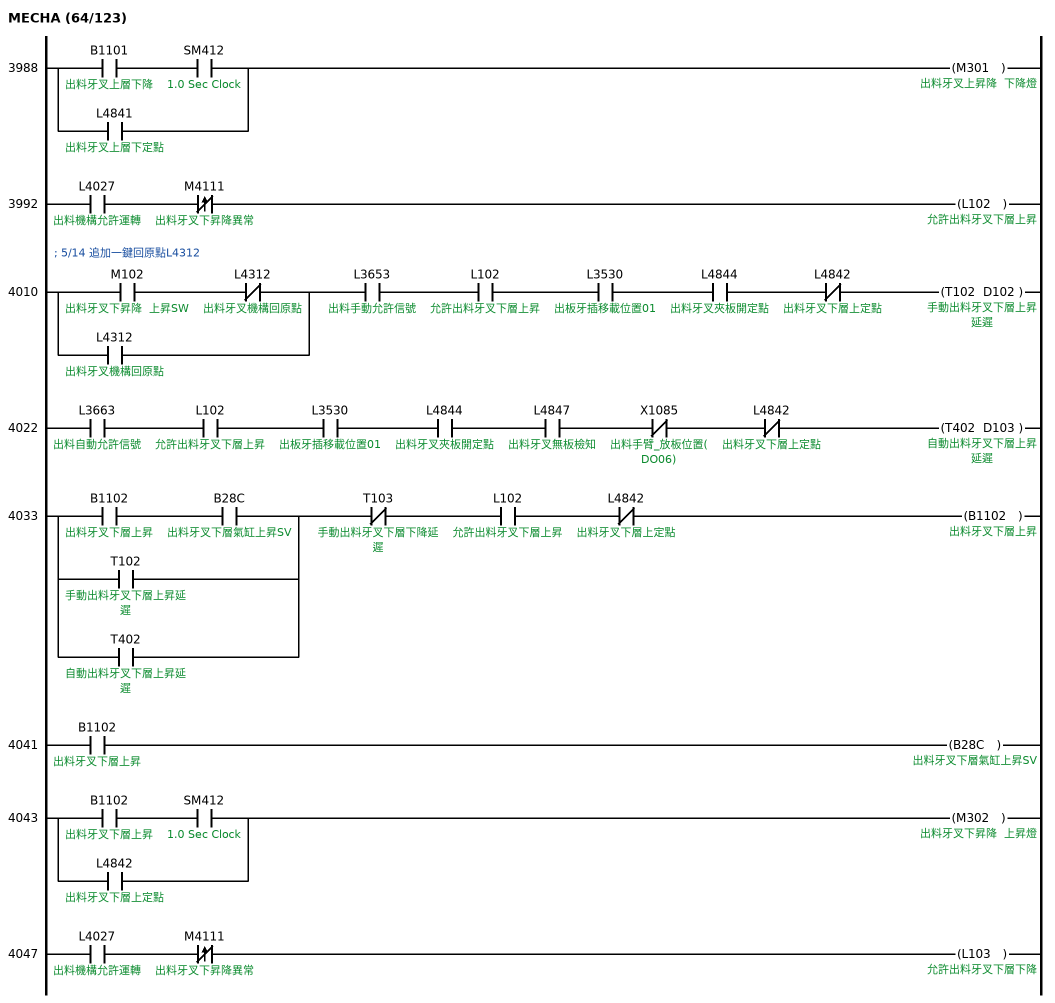
[picture p360: ladder of MECHA, rungs at steps 3988 to 4047]
3988  LD      B1101  ; 出料牙叉上層下降
      AND     SM412  ; 1.0 Sec Clock
      OR      L4841  ; 出料牙叉上層下定點
      OUT     M301  ; 出料牙叉上昇降  下降燈
3992  LD      L4027  ; 出料機構允許運轉
      ANDPI   M4111  ; 出料牙叉下昇降異常
      OUT     L102  ; 允許出料牙叉下層上昇
; 5/14 追加一鍵回原點L4312
4010  LD      M102  ; 出料牙叉下昇降  上昇SW
      ANI     L4312  ; 出料牙叉機構回原點
      OR      L4312  ; 出料牙叉機構回原點
      AND     L3653  ; 出料手動允許信號
      AND     L102  ; 允許出料牙叉下層上昇
      AND     L3530  ; 出板牙插移載位置01
      AND     L4844  ; 出料牙叉夾板開定點
      ANI     L4842  ; 出料牙叉下層上定點
      OUT     T102 D102  ; 手動出料牙叉下層上昇延遲
4022  LD      L3663  ; 出料自動允許信號
      AND     L102  ; 允許出料牙叉下層上昇
      AND     L3530  ; 出板牙插移載位置01
      AND     L4844  ; 出料牙叉夾板開定點
      AND     L4847  ; 出料牙叉無板檢知
      ANI     X1085  ; 出料手臂_放板位置(DO06)
      ANI     L4842  ; 出料牙叉下層上定點
      OUT     T402 D103  ; 自動出料牙叉下層上昇延遲
4033  LD      B1102  ; 出料牙叉下層上昇
      AND     B28C  ; 出料牙叉下層氣缸上昇SV
      OR      T102  ; 手動出料牙叉下層上昇延遲
      OR      T402  ; 自動出料牙叉下層上昇延遲
      ANI     T103  ; 手動出料牙叉下層下降延遲
      AND     L102  ; 允許出料牙叉下層上昇
      ANI     L4842  ; 出料牙叉下層上定點
      OUT     B1102  ; 出料牙叉下層上昇
4041  LD      B1102  ; 出料牙叉下層上昇
      OUT     B28C  ; 出料牙叉下層氣缸上昇SV
4043  LD      B1102  ; 出料牙叉下層上昇
      AND     SM412  ; 1.0 Sec Clock
      OR      L4842  ; 出料牙叉下層上定點
      OUT     M302  ; 出料牙叉下昇降  上昇燈
4047  LD      L4027  ; 出料機構允許運轉
      ANDPI   M4111  ; 出料牙叉下昇降異常
      OUT     L103  ; 允許出料牙叉下層下降
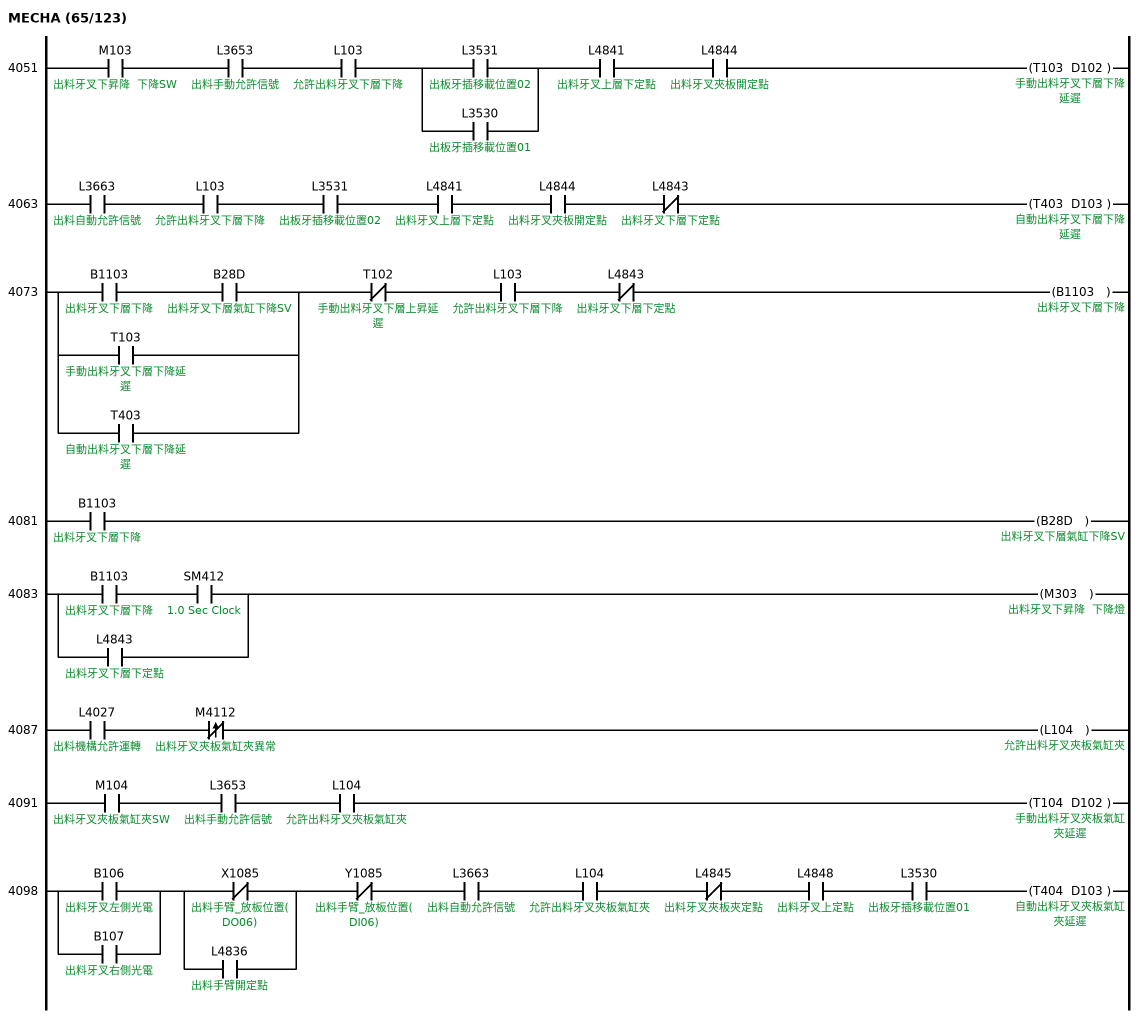
4051  LD      M103  ; 出料牙叉下昇降  下降SW
      AND     L3653  ; 出料手動允許信號
      AND     L103  ; 允許出料牙叉下層下降
      LD      L3531  ; 出板牙插移載位置02
      OR      L3530  ; 出板牙插移載位置01
      ANB
      AND     L4841  ; 出料牙叉上層下定點
      AND     L4844  ; 出料牙叉夾板開定點
      OUT     T103 D102  ; 手動出料牙叉下層下降延遲
4063  LD      L3663  ; 出料自動允許信號
      AND     L103  ; 允許出料牙叉下層下降
      AND     L3531  ; 出板牙插移載位置02
      AND     L4841  ; 出料牙叉上層下定點
      AND     L4844  ; 出料牙叉夾板開定點
      ANI     L4843  ; 出料牙叉下層下定點
      OUT     T403 D103  ; 自動出料牙叉下層下降延遲
4073  LD      B1103  ; 出料牙叉下層下降
      AND     B28D  ; 出料牙叉下層氣缸下降SV
      OR      T103  ; 手動出料牙叉下層下降延遲
      OR      T403  ; 自動出料牙叉下層下降延遲
      ANI     T102  ; 手動出料牙叉下層上昇延遲
      AND     L103  ; 允許出料牙叉下層下降
      ANI     L4843  ; 出料牙叉下層下定點
      OUT     B1103  ; 出料牙叉下層下降
4081  LD      B1103  ; 出料牙叉下層下降
      OUT     B28D  ; 出料牙叉下層氣缸下降SV
4083  LD      B1103  ; 出料牙叉下層下降
      AND     SM412  ; 1.0 Sec Clock
      OR      L4843  ; 出料牙叉下層下定點
      OUT     M303  ; 出料牙叉下昇降  下降燈
4087  LD      L4027  ; 出料機構允許運轉
      ANDPI   M4112  ; 出料牙叉夾板氣缸夾異常
      OUT     L104  ; 允許出料牙叉夾板氣缸夾
4091  LD      M104  ; 出料牙叉夾板氣缸夾SW
      AND     L3653  ; 出料手動允許信號
      AND     L104  ; 允許出料牙叉夾板氣缸夾
      OUT     T104 D102  ; 手動出料牙叉夾板氣缸夾延遲
4098  LD      B106  ; 出料牙叉左側光電
      OR      B107  ; 出料牙叉右側光電
      LDI     X1085  ; 出料手臂_放板位置(DO06)
      OR      L4836  ; 出料手臂開定點
      ANB
      ANI     Y1085  ; 出料手臂_放板位置(DI06)
      AND     L3663  ; 出料自動允許信號
      AND     L104  ; 允許出料牙叉夾板氣缸夾
      ANI     L4845  ; 出料牙叉夾板夾定點
      AND     L4848  ; 出料牙叉上定點
      AND     L3530  ; 出板牙插移載位置01
      OUT     T404 D103  ; 自動出料牙叉夾板氣缸夾延遲
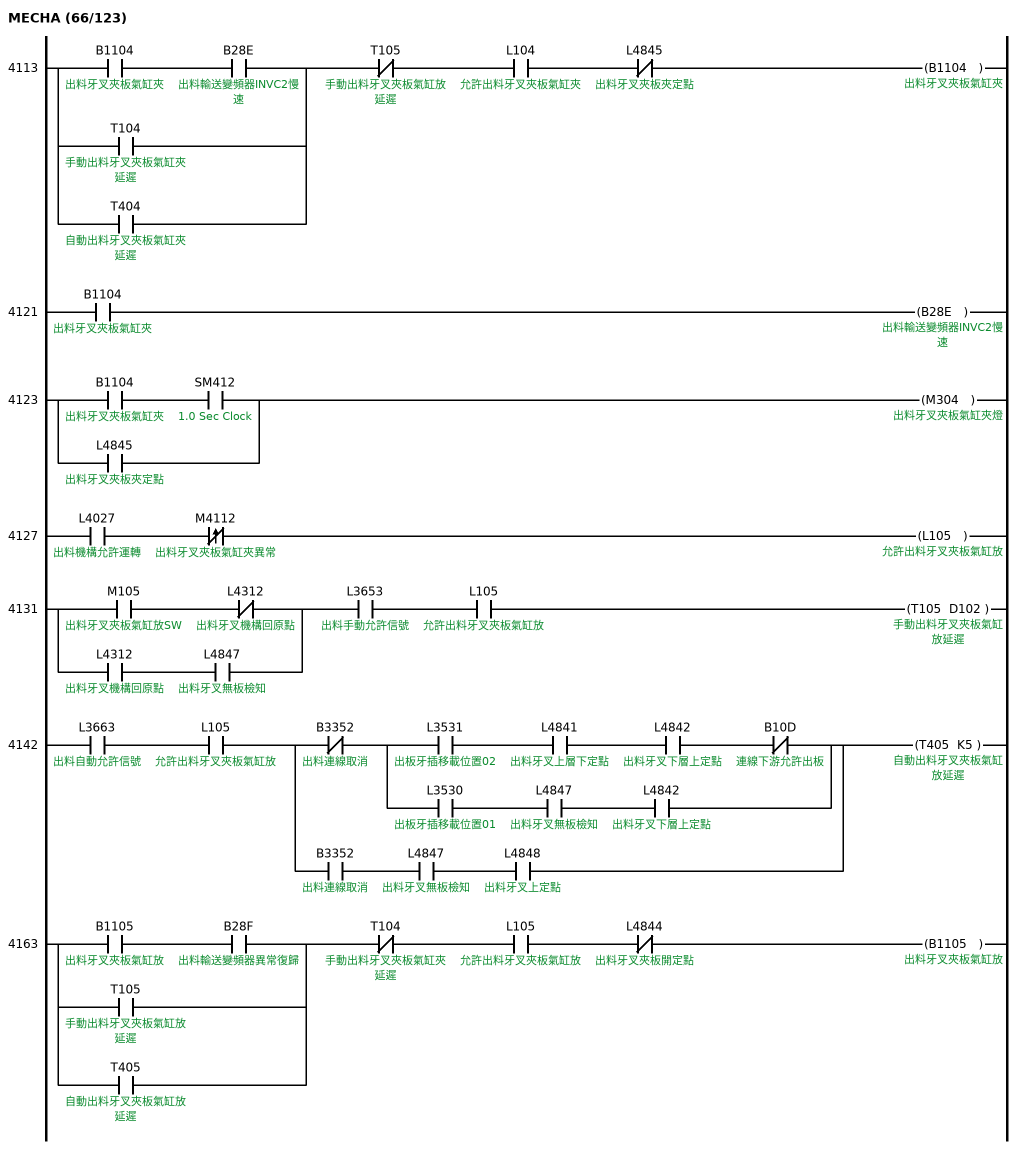
4113  LD      B1104  ; 出料牙叉夾板氣缸夾
      AND     B28E  ; 出料輸送變頻器INVC2慢速
      OR      T104  ; 手動出料牙叉夾板氣缸夾延遲
      OR      T404  ; 自動出料牙叉夾板氣缸夾延遲
      ANI     T105  ; 手動出料牙叉夾板氣缸放延遲
      AND     L104  ; 允許出料牙叉夾板氣缸夾
      ANI     L4845  ; 出料牙叉夾板夾定點
      OUT     B1104  ; 出料牙叉夾板氣缸夾
4121  LD      B1104  ; 出料牙叉夾板氣缸夾
      OUT     B28E  ; 出料輸送變頻器INVC2慢速
4123  LD      B1104  ; 出料牙叉夾板氣缸夾
      AND     SM412  ; 1.0 Sec Clock
      OR      L4845  ; 出料牙叉夾板夾定點
      OUT     M304  ; 出料牙叉夾板氣缸夾燈
4127  LD      L4027  ; 出料機構允許運轉
      ANDPI   M4112  ; 出料牙叉夾板氣缸夾異常
      OUT     L105  ; 允許出料牙叉夾板氣缸放
4131  LD      M105  ; 出料牙叉夾板氣缸放SW
      ANI     L4312  ; 出料牙叉機構回原點
      LD      L4312  ; 出料牙叉機構回原點
      AND     L4847  ; 出料牙叉無板檢知
      ORB
      AND     L3653  ; 出料手動允許信號
      AND     L105  ; 允許出料牙叉夾板氣缸放
      OUT     T105 D102  ; 手動出料牙叉夾板氣缸放延遲
4142  LD      L3663  ; 出料自動允許信號
      AND     L105  ; 允許出料牙叉夾板氣缸放
      LDI     B3352  ; 出料連線取消
      LD      L3531  ; 出板牙插移載位置02
      AND     L4841  ; 出料牙叉上層下定點
      AND     L4842  ; 出料牙叉下層上定點
      ANI     B10D  ; 連線下游允許出板
      LD      L3530  ; 出板牙插移載位置01
      AND     L4847  ; 出料牙叉無板檢知
      AND     L4842  ; 出料牙叉下層上定點
      ORB
      ANB
      LD      B3352  ; 出料連線取消
      AND     L4847  ; 出料牙叉無板檢知
      AND     L4848  ; 出料牙叉上定點
      ORB
      ANB
      OUT     T405 K5  ; 自動出料牙叉夾板氣缸放延遲
4163  LD      B1105  ; 出料牙叉夾板氣缸放
      AND     B28F  ; 出料輸送變頻器異常復歸
      OR      T105  ; 手動出料牙叉夾板氣缸放延遲
      OR      T405  ; 自動出料牙叉夾板氣缸放延遲
      ANI     T104  ; 手動出料牙叉夾板氣缸夾延遲
      AND     L105  ; 允許出料牙叉夾板氣缸放
      ANI     L4844  ; 出料牙叉夾板開定點
      OUT     B1105  ; 出料牙叉夾板氣缸放
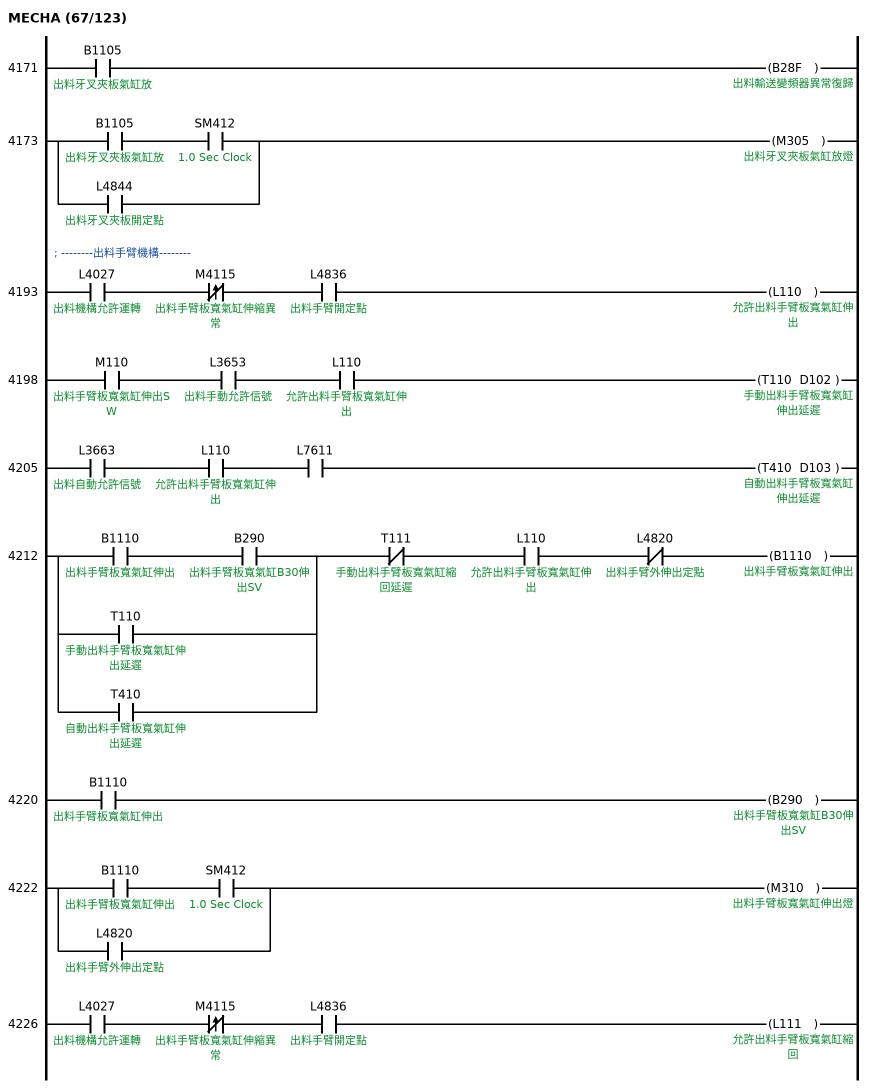
4171  LD      B1105  ; 出料牙叉夾板氣缸放
      OUT     B28F  ; 出料輸送變頻器異常復歸
4173  LD      B1105  ; 出料牙叉夾板氣缸放
      AND     SM412  ; 1.0 Sec Clock
      OR      L4844  ; 出料牙叉夾板開定點
      OUT     M305  ; 出料牙叉夾板氣缸放燈
; --------出料手臂機構--------
4193  LD      L4027  ; 出料機構允許運轉
      ANDPI   M4115  ; 出料手臂板寬氣缸伸縮異常
      AND     L4836  ; 出料手臂開定點
      OUT     L110  ; 允許出料手臂板寬氣缸伸出
4198  LD      M110  ; 出料手臂板寬氣缸伸出SW
      AND     L3653  ; 出料手動允許信號
      AND     L110  ; 允許出料手臂板寬氣缸伸出
      OUT     T110 D102  ; 手動出料手臂板寬氣缸伸出延遲
4205  LD      L3663  ; 出料自動允許信號
      AND     L110  ; 允許出料手臂板寬氣缸伸出
      AND     L7611
      OUT     T410 D103  ; 自動出料手臂板寬氣缸伸出延遲
4212  LD      B1110  ; 出料手臂板寬氣缸伸出
      AND     B290  ; 出料手臂板寬氣缸B30伸出SV
      OR      T110  ; 手動出料手臂板寬氣缸伸出延遲
      OR      T410  ; 自動出料手臂板寬氣缸伸出延遲
      ANI     T111  ; 手動出料手臂板寬氣缸縮回延遲
      AND     L110  ; 允許出料手臂板寬氣缸伸出
      ANI     L4820  ; 出料手臂外伸出定點
      OUT     B1110  ; 出料手臂板寬氣缸伸出
4220  LD      B1110  ; 出料手臂板寬氣缸伸出
      OUT     B290  ; 出料手臂板寬氣缸B30伸出SV
4222  LD      B1110  ; 出料手臂板寬氣缸伸出
      AND     SM412  ; 1.0 Sec Clock
      OR      L4820  ; 出料手臂外伸出定點
      OUT     M310  ; 出料手臂板寬氣缸伸出燈
4226  LD      L4027  ; 出料機構允許運轉
      ANDPI   M4115  ; 出料手臂板寬氣缸伸縮異常
      AND     L4836  ; 出料手臂開定點
      OUT     L111  ; 允許出料手臂板寬氣缸縮回
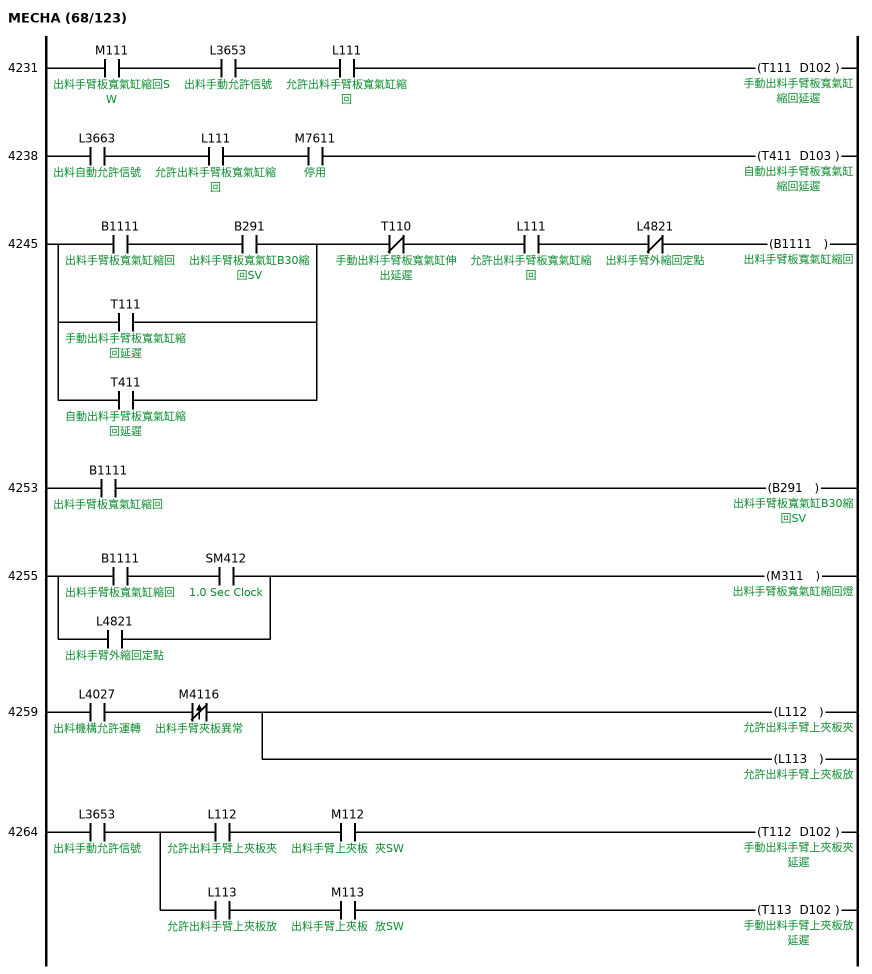
4231  LD      M111  ; 出料手臂板寬氣缸縮回SW
      AND     L3653  ; 出料手動允許信號
      AND     L111  ; 允許出料手臂板寬氣缸縮回
      OUT     T111 D102  ; 手動出料手臂板寬氣缸縮回延遲
4238  LD      L3663  ; 出料自動允許信號
      AND     L111  ; 允許出料手臂板寬氣缸縮回
      AND     M7611  ; 停用
      OUT     T411 D103  ; 自動出料手臂板寬氣缸縮回延遲
4245  LD      B1111  ; 出料手臂板寬氣缸縮回
      AND     B291  ; 出料手臂板寬氣缸B30縮回SV
      OR      T111  ; 手動出料手臂板寬氣缸縮回延遲
      OR      T411  ; 自動出料手臂板寬氣缸縮回延遲
      ANI     T110  ; 手動出料手臂板寬氣缸伸出延遲
      AND     L111  ; 允許出料手臂板寬氣缸縮回
      ANI     L4821  ; 出料手臂外縮回定點
      OUT     B1111  ; 出料手臂板寬氣缸縮回
4253  LD      B1111  ; 出料手臂板寬氣缸縮回
      OUT     B291  ; 出料手臂板寬氣缸B30縮回SV
4255  LD      B1111  ; 出料手臂板寬氣缸縮回
      AND     SM412  ; 1.0 Sec Clock
      OR      L4821  ; 出料手臂外縮回定點
      OUT     M311  ; 出料手臂板寬氣缸縮回燈
4259  LD      L4027  ; 出料機構允許運轉
      ANDPI   M4116  ; 出料手臂夾板異常
      OUT     L112  ; 允許出料手臂上夾板夾
      OUT     L113  ; 允許出料手臂上夾板放
4264  LD      L3653  ; 出料手動允許信號
      MPS
      AND     L112  ; 允許出料手臂上夾板夾
      AND     M112  ; 出料手臂上夾板  夾SW
      OUT     T112 D102  ; 手動出料手臂上夾板夾延遲
      MPP
      AND     L113  ; 允許出料手臂上夾板放
      AND     M113  ; 出料手臂上夾板  放SW
      OUT     T113 D102  ; 手動出料手臂上夾板放延遲
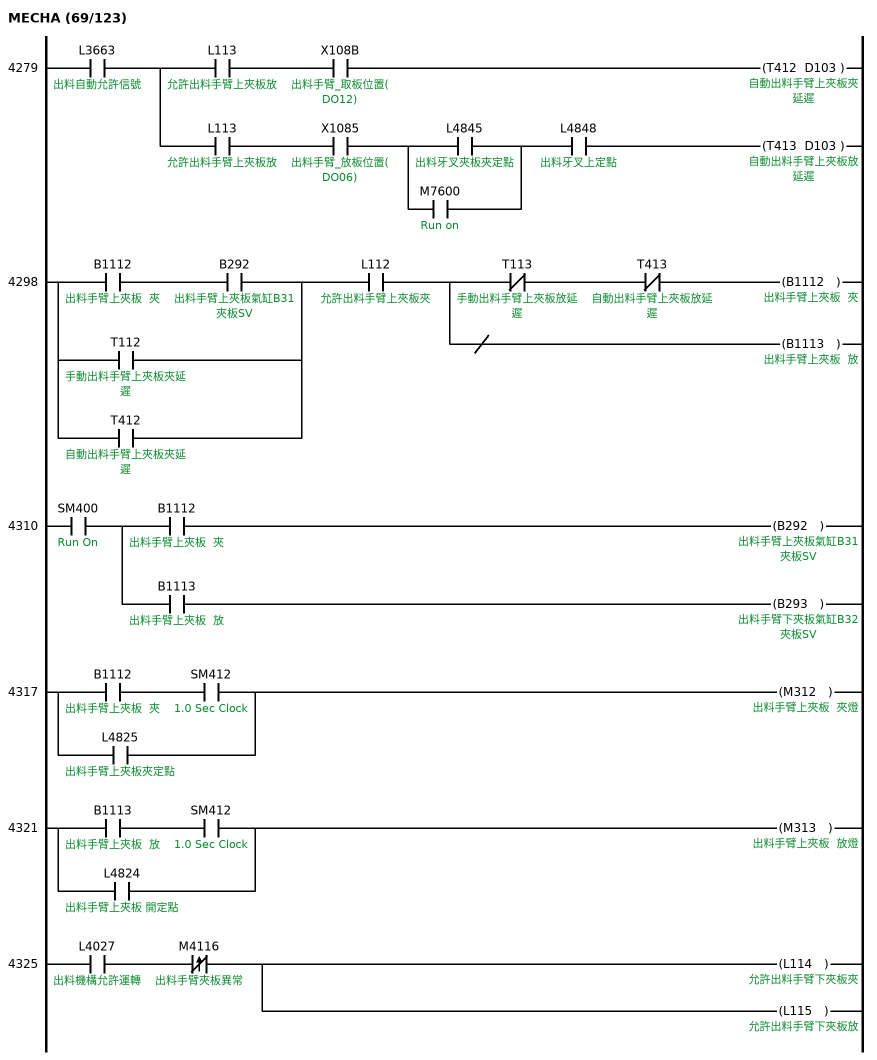
4279  LD      L3663  ; 出料自動允許信號
      MPS
      AND     L113  ; 允許出料手臂上夾板放
      AND     X108B  ; 出料手臂_取板位置(DO12)
      OUT     T412 D103  ; 自動出料手臂上夾板夾延遲
      MPP
      AND     L113  ; 允許出料手臂上夾板放
      AND     X1085  ; 出料手臂_放板位置(DO06)
      LD      L4845  ; 出料牙叉夾板夾定點
      OR      M7600  ; Run on
      ANB
      AND     L4848  ; 出料牙叉上定點
      OUT     T413 D103  ; 自動出料手臂上夾板放延遲
4298  LD      B1112  ; 出料手臂上夾板  夾
      AND     B292  ; 出料手臂上夾板氣缸B31夾板SV
      OR      T112  ; 手動出料手臂上夾板夾延遲
      OR      T412  ; 自動出料手臂上夾板夾延遲
      AND     L112  ; 允許出料手臂上夾板夾
      MPS
      ANI     T113  ; 手動出料手臂上夾板放延遲
      ANI     T413  ; 自動出料手臂上夾板放延遲
      OUT     B1112  ; 出料手臂上夾板  夾
      MPP
      INV
      OUT     B1113  ; 出料手臂上夾板  放
4310  LD      SM400  ; Run On
      MPS
      AND     B1112  ; 出料手臂上夾板  夾
      OUT     B292  ; 出料手臂上夾板氣缸B31夾板SV
      MPP
      AND     B1113  ; 出料手臂上夾板  放
      OUT     B293  ; 出料手臂下夾板氣缸B32夾板SV
4317  LD      B1112  ; 出料手臂上夾板  夾
      AND     SM412  ; 1.0 Sec Clock
      OR      L4825  ; 出料手臂上夾板夾定點
      OUT     M312  ; 出料手臂上夾板  夾燈
4321  LD      B1113  ; 出料手臂上夾板  放
      AND     SM412  ; 1.0 Sec Clock
      OR      L4824  ; 出料手臂上夾板 開定點
      OUT     M313  ; 出料手臂上夾板  放燈
4325  LD      L4027  ; 出料機構允許運轉
      ANDPI   M4116  ; 出料手臂夾板異常
      OUT     L114  ; 允許出料手臂下夾板夾
      OUT     L115  ; 允許出料手臂下夾板放
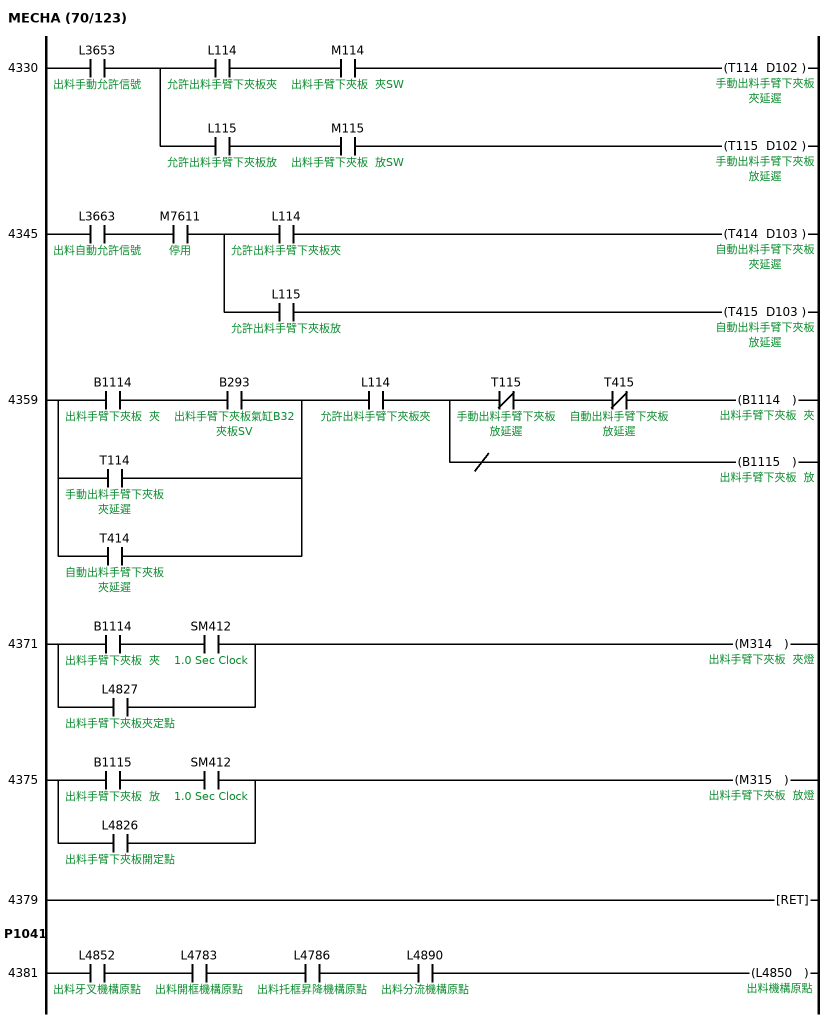
4330  LD      L3653  ; 出料手動允許信號
      MPS
      AND     L114  ; 允許出料手臂下夾板夾
      AND     M114  ; 出料手臂下夾板  夾SW
      OUT     T114 D102  ; 手動出料手臂下夾板  夾延遲
      MPP
      AND     L115  ; 允許出料手臂下夾板放
      AND     M115  ; 出料手臂下夾板  放SW
      OUT     T115 D102  ; 手動出料手臂下夾板  放延遲
4345  LD      L3663  ; 出料自動允許信號
      AND     M7611  ; 停用
      MPS
      AND     L114  ; 允許出料手臂下夾板夾
      OUT     T414 D103  ; 自動出料手臂下夾板  夾延遲
      MPP
      AND     L115  ; 允許出料手臂下夾板放
      OUT     T415 D103  ; 自動出料手臂下夾板  放延遲
4359  LD      B1114  ; 出料手臂下夾板  夾
      AND     B293  ; 出料手臂下夾板氣缸B32夾板SV
      OR      T114  ; 手動出料手臂下夾板  夾延遲
      OR      T414  ; 自動出料手臂下夾板  夾延遲
      AND     L114  ; 允許出料手臂下夾板夾
      MPS
      ANI     T115  ; 手動出料手臂下夾板  放延遲
      ANI     T415  ; 自動出料手臂下夾板  放延遲
      OUT     B1114  ; 出料手臂下夾板  夾
      MPP
      INV
      OUT     B1115  ; 出料手臂下夾板  放
4371  LD      B1114  ; 出料手臂下夾板  夾
      AND     SM412  ; 1.0 Sec Clock
      OR      L4827  ; 出料手臂下夾板夾定點
      OUT     M314  ; 出料手臂下夾板  夾燈
4375  LD      B1115  ; 出料手臂下夾板  放
      AND     SM412  ; 1.0 Sec Clock
      OR      L4826  ; 出料手臂下夾板開定點
      OUT     M315  ; 出料手臂下夾板  放燈
4379  RET
      P1041
4381  LD      L4852  ; 出料牙叉機構原點
      AND     L4783  ; 出料開框機構原點
      AND     L4786  ; 出料托框昇降機構原點
      AND     L4890  ; 出料分流機構原點
      OUT     L4850  ; 出料機構原點
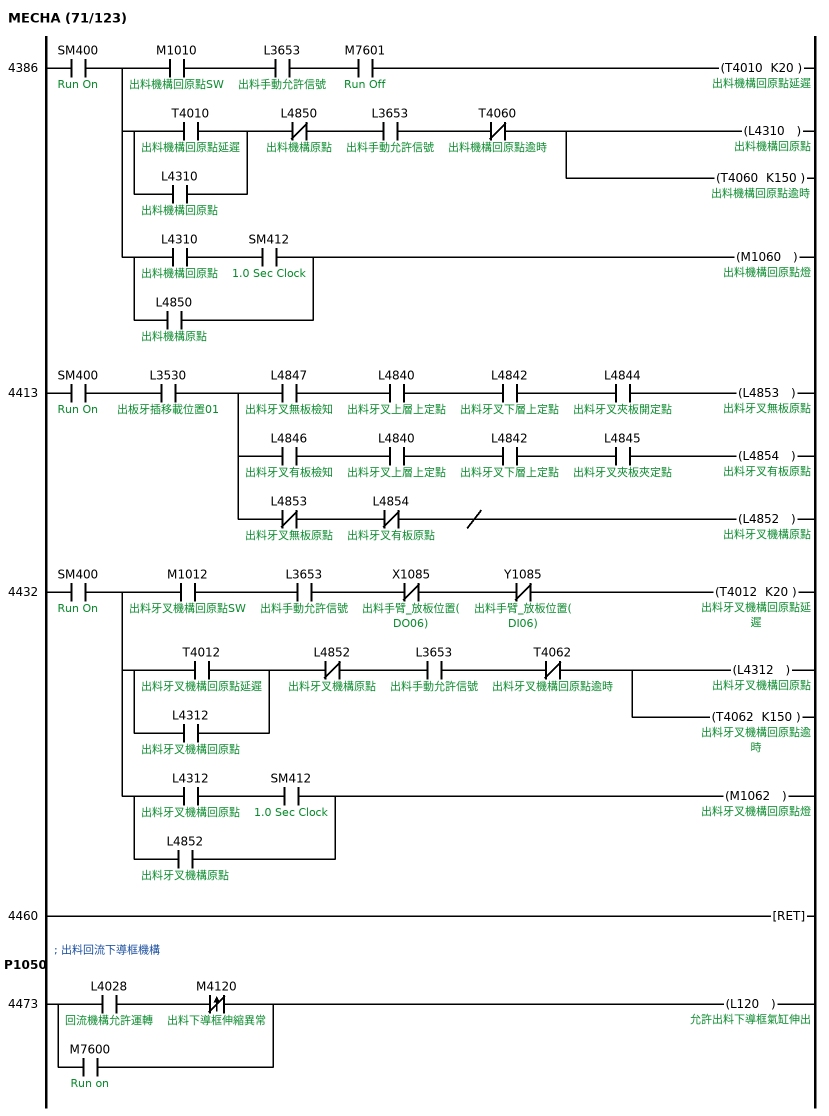
4386  LD      SM400  ; Run On
      MPS
      AND     M1010  ; 出料機構回原點SW
      AND     L3653  ; 出料手動允許信號
      AND     M7601  ; Run Off
      OUT     T4010 K20  ; 出料機構回原點延遲
      MRD
      LD      T4010  ; 出料機構回原點延遲
      OR      L4310  ; 出料機構回原點
      ANB
      ANI     L4850  ; 出料機構原點
      AND     L3653  ; 出料手動允許信號
      ANI     T4060  ; 出料機構回原點逾時
      OUT     L4310  ; 出料機構回原點
      OUT     T4060 K150  ; 出料機構回原點逾時
      MPP
      LD      L4310  ; 出料機構回原點
      AND     SM412  ; 1.0 Sec Clock
      OR      L4850  ; 出料機構原點
      ANB
      OUT     M1060  ; 出料機構回原點燈
4413  LD      SM400  ; Run On
      AND     L3530  ; 出板牙插移載位置01
      MPS
      AND     L4847  ; 出料牙叉無板檢知
      AND     L4840  ; 出料牙叉上層上定點
      AND     L4842  ; 出料牙叉下層上定點
      AND     L4844  ; 出料牙叉夾板開定點
      OUT     L4853  ; 出料牙叉無板原點
      MRD
      AND     L4846  ; 出料牙叉有板檢知
      AND     L4840  ; 出料牙叉上層上定點
      AND     L4842  ; 出料牙叉下層上定點
      AND     L4845  ; 出料牙叉夾板夾定點
      OUT     L4854  ; 出料牙叉有板原點
      MPP
      ANI     L4853  ; 出料牙叉無板原點
      ANI     L4854  ; 出料牙叉有板原點
      INV
      OUT     L4852  ; 出料牙叉機構原點
4432  LD      SM400  ; Run On
      MPS
      AND     M1012  ; 出料牙叉機構回原點SW
      AND     L3653  ; 出料手動允許信號
      ANI     X1085  ; 出料手臂_放板位置(DO06)
      ANI     Y1085  ; 出料手臂_放板位置(DI06)
      OUT     T4012 K20  ; 出料牙叉機構回原點延遲
      MRD
      LD      T4012  ; 出料牙叉機構回原點延遲
      OR      L4312  ; 出料牙叉機構回原點
      ANB
      ANI     L4852  ; 出料牙叉機構原點
      AND     L3653  ; 出料手動允許信號
      ANI     T4062  ; 出料牙叉機構回原點逾時
      OUT     L4312  ; 出料牙叉機構回原點
      OUT     T4062 K150  ; 出料牙叉機構回原點逾時
      MPP
      LD      L4312  ; 出料牙叉機構回原點
      AND     SM412  ; 1.0 Sec Clock
      OR      L4852  ; 出料牙叉機構原點
      ANB
      OUT     M1062  ; 出料牙叉機構回原點燈
4460  RET
; 出料回流下導框機構
      P1050
4473  LD      L4028  ; 回流機構允許運轉
      ANDPI   M4120  ; 出料下導框伸縮異常
      OR      M7600  ; Run on
      OUT     L120  ; 允許出料下導框氣缸伸出
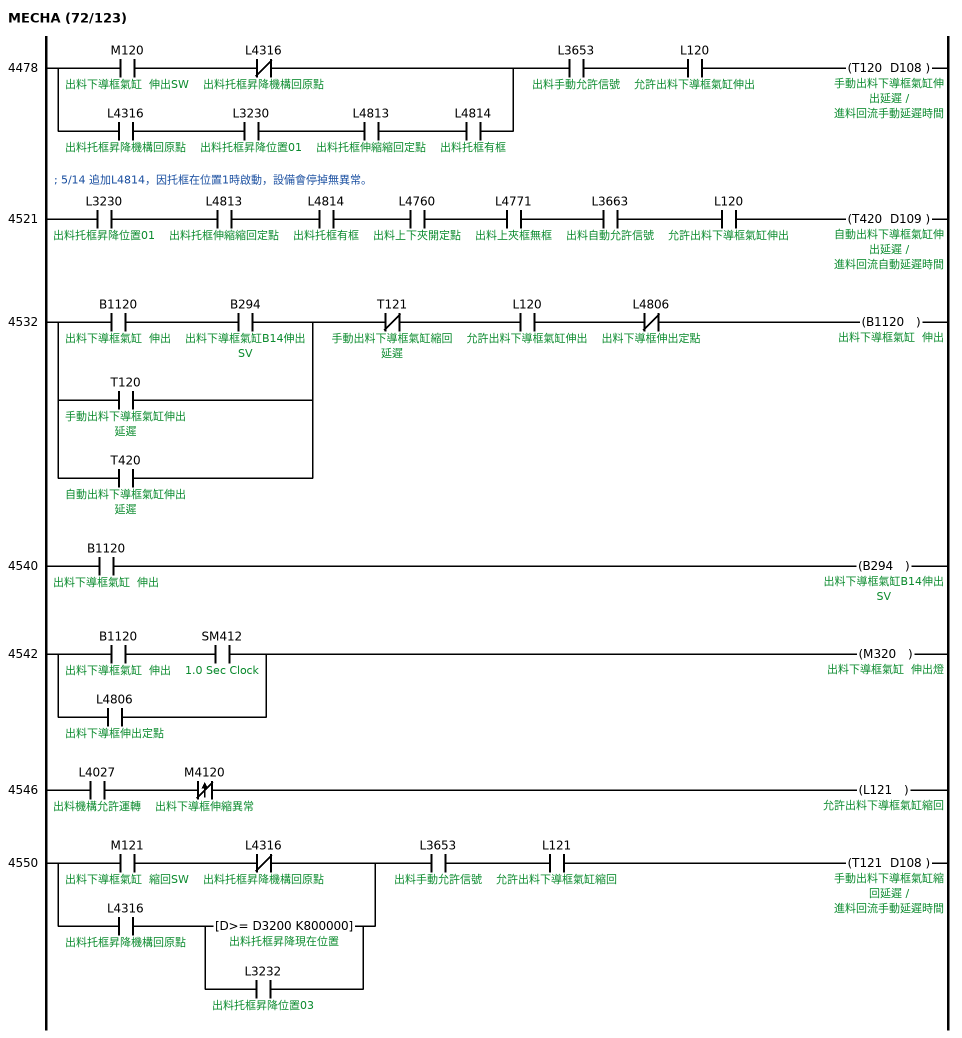
4478  LD      M120  ; 出料下導框氣缸  伸出SW
      ANI     L4316  ; 出料托框昇降機構回原點
      LD      L4316  ; 出料托框昇降機構回原點
      AND     L3230  ; 出料托框昇降位置01
      AND     L4813  ; 出料托框伸縮縮回定點
      AND     L4814  ; 出料托框有框
      ORB
      AND     L3653  ; 出料手動允許信號
      AND     L120  ; 允許出料下導框氣缸伸出
      OUT     T120 D108  ; 手動出料下導框氣缸伸出延遲 / 進料回流手動延遲時間
; 5/14 追加L4814，因托框在位置1時啟動，設備會停掉無異常。
4521  LD      L3230  ; 出料托框昇降位置01
      AND     L4813  ; 出料托框伸縮縮回定點
      AND     L4814  ; 出料托框有框
      AND     L4760  ; 出料上下夾開定點
      AND     L4771  ; 出料上夾框無框
      AND     L3663  ; 出料自動允許信號
      AND     L120  ; 允許出料下導框氣缸伸出
      OUT     T420 D109  ; 自動出料下導框氣缸伸出延遲 / 進料回流自動延遲時間
4532  LD      B1120  ; 出料下導框氣缸  伸出
      AND     B294  ; 出料下導框氣缸B14伸出SV
      OR      T120  ; 手動出料下導框氣缸伸出延遲
      OR      T420  ; 自動出料下導框氣缸伸出延遲
      ANI     T121  ; 手動出料下導框氣缸縮回延遲
      AND     L120  ; 允許出料下導框氣缸伸出
      ANI     L4806  ; 出料下導框伸出定點
      OUT     B1120  ; 出料下導框氣缸  伸出
4540  LD      B1120  ; 出料下導框氣缸  伸出
      OUT     B294  ; 出料下導框氣缸B14伸出SV
4542  LD      B1120  ; 出料下導框氣缸  伸出
      AND     SM412  ; 1.0 Sec Clock
      OR      L4806  ; 出料下導框伸出定點
      OUT     M320  ; 出料下導框氣缸  伸出燈
4546  LD      L4027  ; 出料機構允許運轉
      ANDPI   M4120  ; 出料下導框伸縮異常
      OUT     L121  ; 允許出料下導框氣缸縮回
4550  LD      M121  ; 出料下導框氣缸  縮回SW
      ANI     L4316  ; 出料托框昇降機構回原點
      LD      L4316  ; 出料托框昇降機構回原點
      LDD>=   D3200 K800000  ; 出料托框昇降現在位置
      OR      L3232  ; 出料托框昇降位置03
      ANB
      ORB
      AND     L3653  ; 出料手動允許信號
      AND     L121  ; 允許出料下導框氣缸縮回
      OUT     T121 D108  ; 手動出料下導框氣缸縮回延遲 / 進料回流手動延遲時間
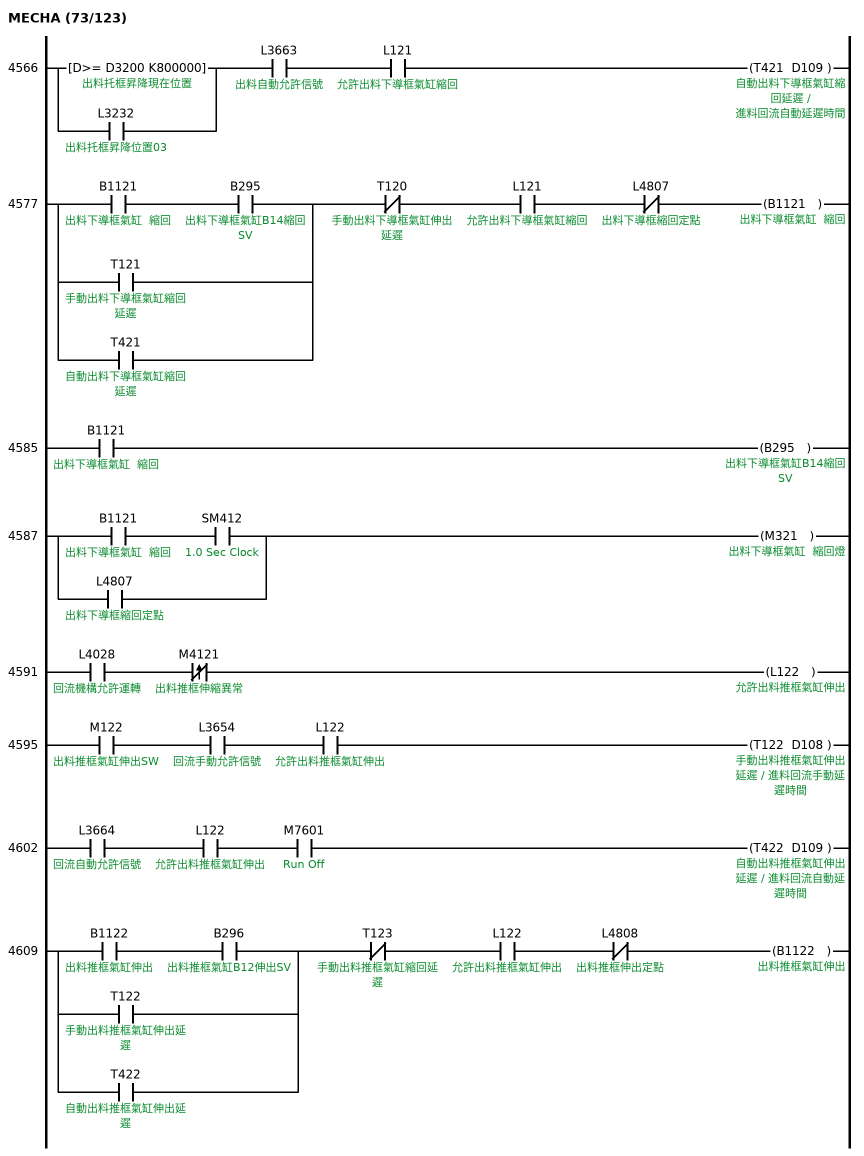
4566  LDD>=   D3200 K800000  ; 出料托框昇降現在位置
      OR      L3232  ; 出料托框昇降位置03
      AND     L3663  ; 出料自動允許信號
      AND     L121  ; 允許出料下導框氣缸縮回
      OUT     T421 D109  ; 自動出料下導框氣缸縮回延遲 / 進料回流自動延遲時間
4577  LD      B1121  ; 出料下導框氣缸  縮回
      AND     B295  ; 出料下導框氣缸B14縮回SV
      OR      T121  ; 手動出料下導框氣缸縮回延遲
      OR      T421  ; 自動出料下導框氣缸縮回延遲
      ANI     T120  ; 手動出料下導框氣缸伸出延遲
      AND     L121  ; 允許出料下導框氣缸縮回
      ANI     L4807  ; 出料下導框縮回定點
      OUT     B1121  ; 出料下導框氣缸  縮回
4585  LD      B1121  ; 出料下導框氣缸  縮回
      OUT     B295  ; 出料下導框氣缸B14縮回SV
4587  LD      B1121  ; 出料下導框氣缸  縮回
      AND     SM412  ; 1.0 Sec Clock
      OR      L4807  ; 出料下導框縮回定點
      OUT     M321  ; 出料下導框氣缸  縮回燈
4591  LD      L4028  ; 回流機構允許運轉
      ANDPI   M4121  ; 出料推框伸縮異常
      OUT     L122  ; 允許出料推框氣缸伸出
4595  LD      M122  ; 出料推框氣缸伸出SW
      AND     L3654  ; 回流手動允許信號
      AND     L122  ; 允許出料推框氣缸伸出
      OUT     T122 D108  ; 手動出料推框氣缸伸出延遲 / 進料回流手動延遲時間
4602  LD      L3664  ; 回流自動允許信號
      AND     L122  ; 允許出料推框氣缸伸出
      AND     M7601  ; Run Off
      OUT     T422 D109  ; 自動出料推框氣缸伸出延遲 / 進料回流自動延遲時間
4609  LD      B1122  ; 出料推框氣缸伸出
      AND     B296  ; 出料推框氣缸B12伸出SV
      OR      T122  ; 手動出料推框氣缸伸出延遲
      OR      T422  ; 自動出料推框氣缸伸出延遲
      ANI     T123  ; 手動出料推框氣缸縮回延遲
      AND     L122  ; 允許出料推框氣缸伸出
      ANI     L4808  ; 出料推框伸出定點
      OUT     B1122  ; 出料推框氣缸伸出
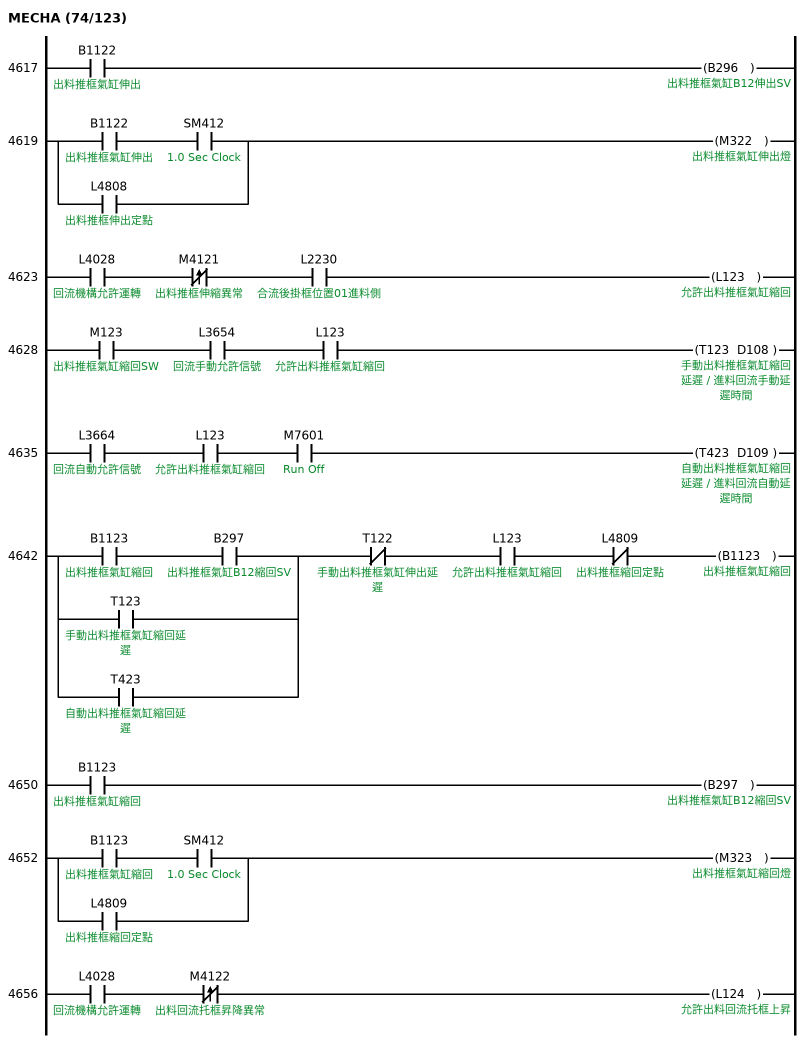
4617  LD      B1122  ; 出料推框氣缸伸出
      OUT     B296  ; 出料推框氣缸B12伸出SV
4619  LD      B1122  ; 出料推框氣缸伸出
      AND     SM412  ; 1.0 Sec Clock
      OR      L4808  ; 出料推框伸出定點
      OUT     M322  ; 出料推框氣缸伸出燈
4623  LD      L4028  ; 回流機構允許運轉
      ANDPI   M4121  ; 出料推框伸縮異常
      AND     L2230  ; 合流後掛框位置01進料側
      OUT     L123  ; 允許出料推框氣缸縮回
4628  LD      M123  ; 出料推框氣缸縮回SW
      AND     L3654  ; 回流手動允許信號
      AND     L123  ; 允許出料推框氣缸縮回
      OUT     T123 D108  ; 手動出料推框氣缸縮回延遲 / 進料回流手動延遲時間
4635  LD      L3664  ; 回流自動允許信號
      AND     L123  ; 允許出料推框氣缸縮回
      AND     M7601  ; Run Off
      OUT     T423 D109  ; 自動出料推框氣缸縮回延遲 / 進料回流自動延遲時間
4642  LD      B1123  ; 出料推框氣缸縮回
      AND     B297  ; 出料推框氣缸B12縮回SV
      OR      T123  ; 手動出料推框氣缸縮回延遲
      OR      T423  ; 自動出料推框氣缸縮回延遲
      ANI     T122  ; 手動出料推框氣缸伸出延遲
      AND     L123  ; 允許出料推框氣缸縮回
      ANI     L4809  ; 出料推框縮回定點
      OUT     B1123  ; 出料推框氣缸縮回
4650  LD      B1123  ; 出料推框氣缸縮回
      OUT     B297  ; 出料推框氣缸B12縮回SV
4652  LD      B1123  ; 出料推框氣缸縮回
      AND     SM412  ; 1.0 Sec Clock
      OR      L4809  ; 出料推框縮回定點
      OUT     M323  ; 出料推框氣缸縮回燈
4656  LD      L4028  ; 回流機構允許運轉
      ANDPI   M4122  ; 出料回流托框昇降異常
      OUT     L124  ; 允許出料回流托框上昇
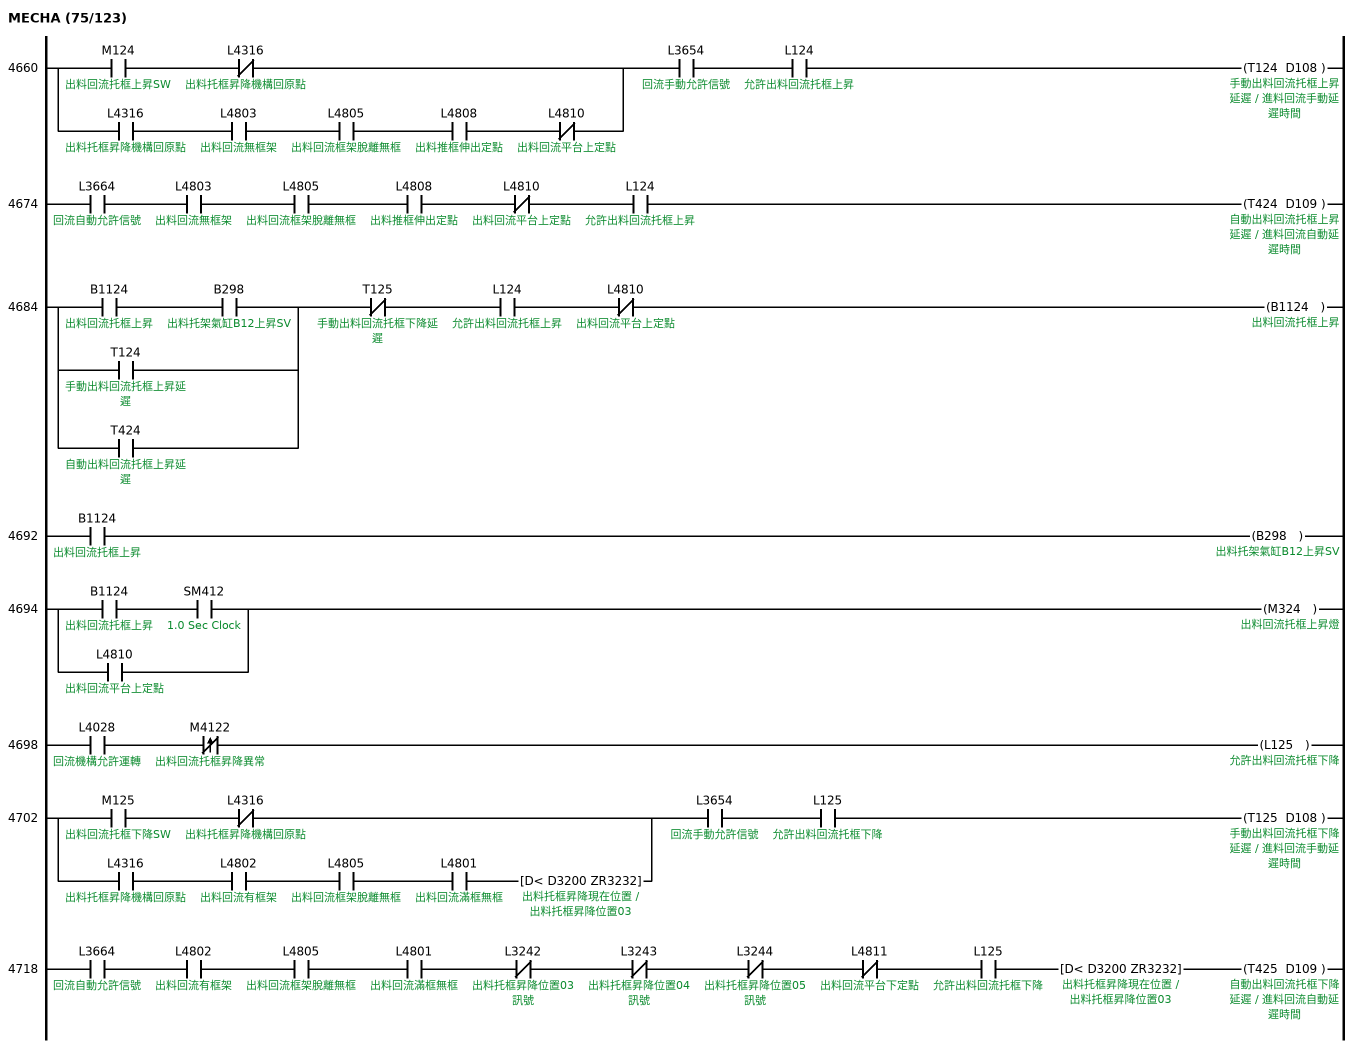
4660  LD      M124  ; 出料回流托框上昇SW
      ANI     L4316  ; 出料托框昇降機構回原點
      LD      L4316  ; 出料托框昇降機構回原點
      AND     L4803  ; 出料回流無框架
      AND     L4805  ; 出料回流框架脫離無框
      AND     L4808  ; 出料推框伸出定點
      ANI     L4810  ; 出料回流平台上定點
      ORB
      AND     L3654  ; 回流手動允許信號
      AND     L124  ; 允許出料回流托框上昇
      OUT     T124 D108  ; 手動出料回流托框上昇延遲 / 進料回流手動延遲時間
4674  LD      L3664  ; 回流自動允許信號
      AND     L4803  ; 出料回流無框架
      AND     L4805  ; 出料回流框架脫離無框
      AND     L4808  ; 出料推框伸出定點
      ANI     L4810  ; 出料回流平台上定點
      AND     L124  ; 允許出料回流托框上昇
      OUT     T424 D109  ; 自動出料回流托框上昇延遲 / 進料回流自動延遲時間
4684  LD      B1124  ; 出料回流托框上昇
      AND     B298  ; 出料托架氣缸B12上昇SV
      OR      T124  ; 手動出料回流托框上昇延遲
      OR      T424  ; 自動出料回流托框上昇延遲
      ANI     T125  ; 手動出料回流托框下降延遲
      AND     L124  ; 允許出料回流托框上昇
      ANI     L4810  ; 出料回流平台上定點
      OUT     B1124  ; 出料回流托框上昇
4692  LD      B1124  ; 出料回流托框上昇
      OUT     B298  ; 出料托架氣缸B12上昇SV
4694  LD      B1124  ; 出料回流托框上昇
      AND     SM412  ; 1.0 Sec Clock
      OR      L4810  ; 出料回流平台上定點
      OUT     M324  ; 出料回流托框上昇燈
4698  LD      L4028  ; 回流機構允許運轉
      ANDPI   M4122  ; 出料回流托框昇降異常
      OUT     L125  ; 允許出料回流托框下降
4702  LD      M125  ; 出料回流托框下降SW
      ANI     L4316  ; 出料托框昇降機構回原點
      LD      L4316  ; 出料托框昇降機構回原點
      AND     L4802  ; 出料回流有框架
      AND     L4805  ; 出料回流框架脫離無框
      AND     L4801  ; 出料回流滿框無框
      ANDD<   D3200 ZR3232  ; 出料托框昇降現在位置 / 出料托框昇降位置03
      ORB
      AND     L3654  ; 回流手動允許信號
      AND     L125  ; 允許出料回流托框下降
      OUT     T125 D108  ; 手動出料回流托框下降延遲 / 進料回流手動延遲時間
4718  LD      L3664  ; 回流自動允許信號
      AND     L4802  ; 出料回流有框架
      AND     L4805  ; 出料回流框架脫離無框
      AND     L4801  ; 出料回流滿框無框
      ANI     L3242  ; 出料托框昇降位置03 訊號
      ANI     L3243  ; 出料托框昇降位置04 訊號
      ANI     L3244  ; 出料托框昇降位置05 訊號
      ANI     L4811  ; 出料回流平台下定點
      AND     L125  ; 允許出料回流托框下降
      ANDD<   D3200 ZR3232  ; 出料托框昇降現在位置 / 出料托框昇降位置03
      OUT     T425 D109  ; 自動出料回流托框下降延遲 / 進料回流自動延遲時間
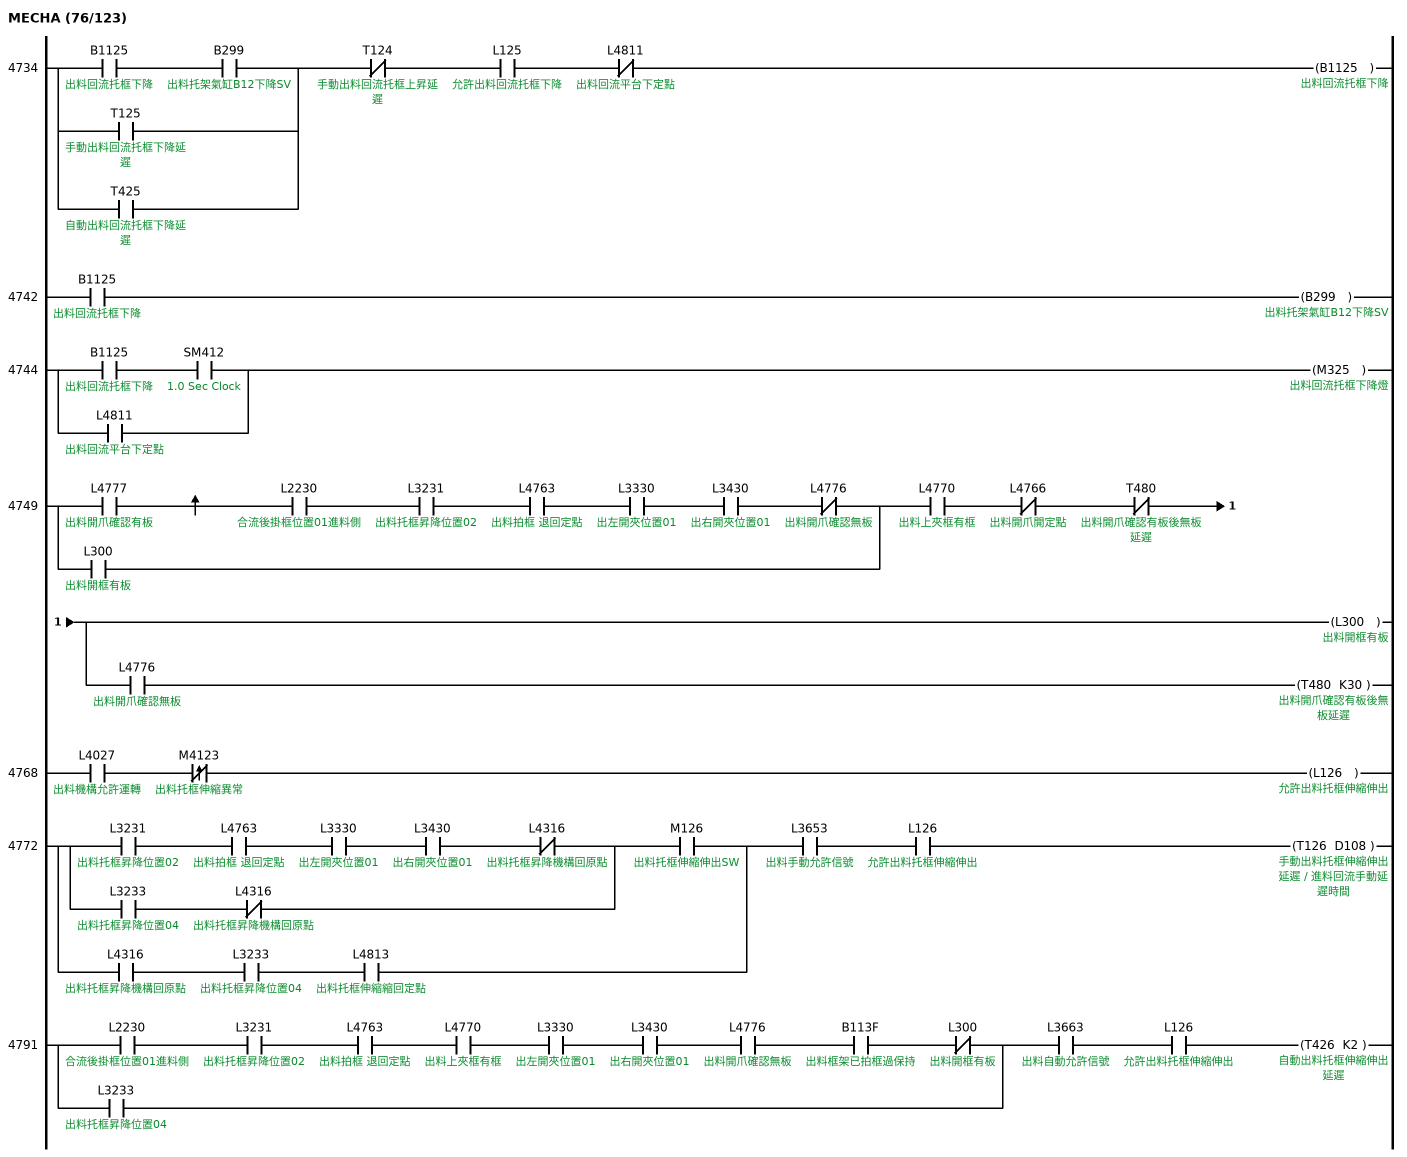
4734  LD      B1125  ; 出料回流托框下降
      AND     B299  ; 出料托架氣缸B12下降SV
      OR      T125  ; 手動出料回流托框下降延遲
      OR      T425  ; 自動出料回流托框下降延遲
      ANI     T124  ; 手動出料回流托框上昇延遲
      AND     L125  ; 允許出料回流托框下降
      ANI     L4811  ; 出料回流平台下定點
      OUT     B1125  ; 出料回流托框下降
4742  LD      B1125  ; 出料回流托框下降
      OUT     B299  ; 出料托架氣缸B12下降SV
4744  LD      B1125  ; 出料回流托框下降
      AND     SM412  ; 1.0 Sec Clock
      OR      L4811  ; 出料回流平台下定點
      OUT     M325  ; 出料回流托框下降燈
4749  LD      L4777  ; 出料開爪確認有板
      MEP
      AND     L2230  ; 合流後掛框位置01進料側
      AND     L3231  ; 出料托框昇降位置02
      AND     L4763  ; 出料拍框 退回定點
      AND     L3330  ; 出左開夾位置01
      AND     L3430  ; 出右開夾位置01
      ANI     L4776  ; 出料開爪確認無板
      OR      L300  ; 出料開框有板
      AND     L4770  ; 出料上夾框有框
      ANI     L4766  ; 出料開爪開定點
      ANI     T480  ; 出料開爪確認有板後無板延遲
      OUT     L300  ; 出料開框有板
      AND     L4776  ; 出料開爪確認無板
      OUT     T480 K30  ; 出料開爪確認有板後無板延遲
4768  LD      L4027  ; 出料機構允許運轉
      ANDPI   M4123  ; 出料托框伸縮異常
      OUT     L126  ; 允許出料托框伸縮伸出
4772  LD      L3231  ; 出料托框昇降位置02
      AND     L4763  ; 出料拍框 退回定點
      AND     L3330  ; 出左開夾位置01
      AND     L3430  ; 出右開夾位置01
      ANI     L4316  ; 出料托框昇降機構回原點
      LD      L3233  ; 出料托框昇降位置04
      ANI     L4316  ; 出料托框昇降機構回原點
      ORB
      AND     M126  ; 出料托框伸縮伸出SW
      LD      L4316  ; 出料托框昇降機構回原點
      AND     L3233  ; 出料托框昇降位置04
      AND     L4813  ; 出料托框伸縮縮回定點
      ORB
      AND     L3653  ; 出料手動允許信號
      AND     L126  ; 允許出料托框伸縮伸出
      OUT     T126 D108  ; 手動出料托框伸縮伸出延遲 / 進料回流手動延遲時間
4791  LD      L2230  ; 合流後掛框位置01進料側
      AND     L3231  ; 出料托框昇降位置02
      AND     L4763  ; 出料拍框 退回定點
      AND     L4770  ; 出料上夾框有框
      AND     L3330  ; 出左開夾位置01
      AND     L3430  ; 出右開夾位置01
      AND     L4776  ; 出料開爪確認無板
      AND     B113F  ; 出料框架已拍框過保持
      ANI     L300  ; 出料開框有板
      OR      L3233  ; 出料托框昇降位置04
      AND     L3663  ; 出料自動允許信號
      AND     L126  ; 允許出料托框伸縮伸出
      OUT     T426 K2  ; 自動出料托框伸縮伸出延遲
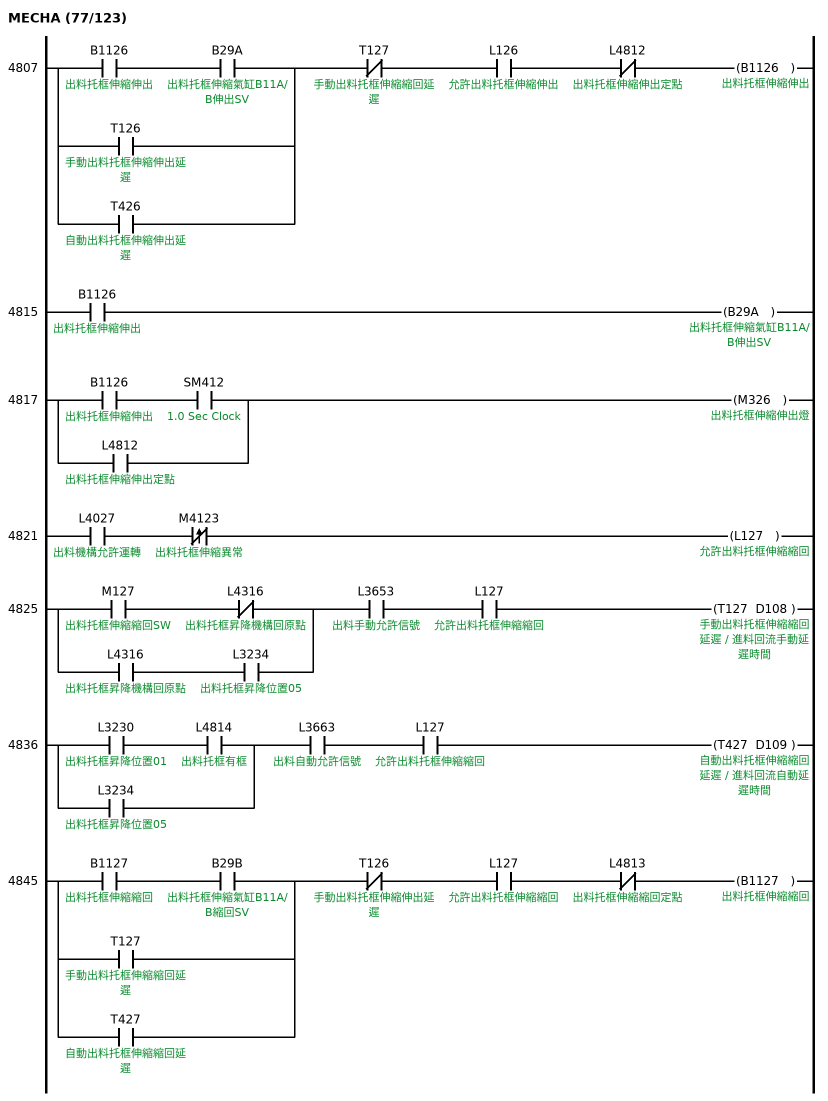
4807  LD      B1126  ; 出料托框伸縮伸出
      AND     B29A  ; 出料托框伸縮氣缸B11A/B伸出SV
      OR      T126  ; 手動出料托框伸縮伸出延遲
      OR      T426  ; 自動出料托框伸縮伸出延遲
      ANI     T127  ; 手動出料托框伸縮縮回延遲
      AND     L126  ; 允許出料托框伸縮伸出
      ANI     L4812  ; 出料托框伸縮伸出定點
      OUT     B1126  ; 出料托框伸縮伸出
4815  LD      B1126  ; 出料托框伸縮伸出
      OUT     B29A  ; 出料托框伸縮氣缸B11A/B伸出SV
4817  LD      B1126  ; 出料托框伸縮伸出
      AND     SM412  ; 1.0 Sec Clock
      OR      L4812  ; 出料托框伸縮伸出定點
      OUT     M326  ; 出料托框伸縮伸出燈
4821  LD      L4027  ; 出料機構允許運轉
      ANDPI   M4123  ; 出料托框伸縮異常
      OUT     L127  ; 允許出料托框伸縮縮回
4825  LD      M127  ; 出料托框伸縮縮回SW
      ANI     L4316  ; 出料托框昇降機構回原點
      LD      L4316  ; 出料托框昇降機構回原點
      AND     L3234  ; 出料托框昇降位置05
      ORB
      AND     L3653  ; 出料手動允許信號
      AND     L127  ; 允許出料托框伸縮縮回
      OUT     T127 D108  ; 手動出料托框伸縮縮回延遲 / 進料回流手動延遲時間
4836  LD      L3230  ; 出料托框昇降位置01
      AND     L4814  ; 出料托框有框
      OR      L3234  ; 出料托框昇降位置05
      AND     L3663  ; 出料自動允許信號
      AND     L127  ; 允許出料托框伸縮縮回
      OUT     T427 D109  ; 自動出料托框伸縮縮回延遲 / 進料回流自動延遲時間
4845  LD      B1127  ; 出料托框伸縮縮回
      AND     B29B  ; 出料托框伸縮氣缸B11A/B縮回SV
      OR      T127  ; 手動出料托框伸縮縮回延遲
      OR      T427  ; 自動出料托框伸縮縮回延遲
      ANI     T126  ; 手動出料托框伸縮伸出延遲
      AND     L127  ; 允許出料托框伸縮縮回
      ANI     L4813  ; 出料托框伸縮縮回定點
      OUT     B1127  ; 出料托框伸縮縮回
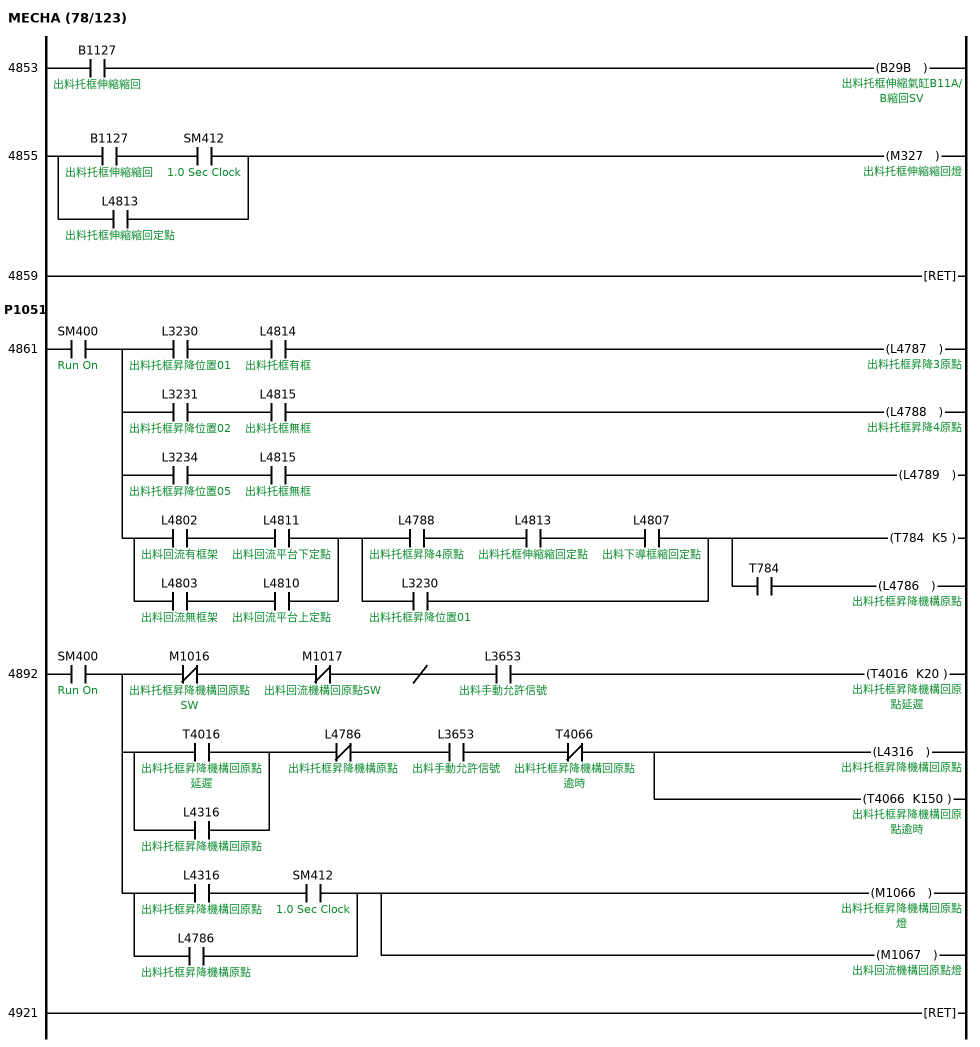
4853  LD      B1127  ; 出料托框伸縮縮回
      OUT     B29B  ; 出料托框伸縮氣缸B11A/B縮回SV
4855  LD      B1127  ; 出料托框伸縮縮回
      AND     SM412  ; 1.0 Sec Clock
      OR      L4813  ; 出料托框伸縮縮回定點
      OUT     M327  ; 出料托框伸縮縮回燈
4859  RET
      P1051
4861  LD      SM400  ; Run On
      MPS
      AND     L3230  ; 出料托框昇降位置01
      AND     L4814  ; 出料托框有框
      OUT     L4787  ; 出料托框昇降3原點
      MRD
      AND     L3231  ; 出料托框昇降位置02
      AND     L4815  ; 出料托框無框
      OUT     L4788  ; 出料托框昇降4原點
      MRD
      AND     L3234  ; 出料托框昇降位置05
      AND     L4815  ; 出料托框無框
      OUT     L4789
      MPP
      LD      L4802  ; 出料回流有框架
      AND     L4811  ; 出料回流平台下定點
      LD      L4803  ; 出料回流無框架
      AND     L4810  ; 出料回流平台上定點
      ORB
      ANB
      LD      L4788  ; 出料托框昇降4原點
      AND     L4813  ; 出料托框伸縮縮回定點
      AND     L4807  ; 出料下導框縮回定點
      OR      L3230  ; 出料托框昇降位置01
      ANB
      OUT     T784 K5
      AND     T784
      OUT     L4786  ; 出料托框昇降機構原點
4892  LD      SM400  ; Run On
      MPS
      ANI     M1016  ; 出料托框昇降機構回原點SW
      ANI     M1017  ; 出料回流機構回原點SW
      INV
      AND     L3653  ; 出料手動允許信號
      OUT     T4016 K20  ; 出料托框昇降機構回原點延遲
      MRD
      LD      T4016  ; 出料托框昇降機構回原點延遲
      OR      L4316  ; 出料托框昇降機構回原點
      ANB
      ANI     L4786  ; 出料托框昇降機構原點
      AND     L3653  ; 出料手動允許信號
      ANI     T4066  ; 出料托框昇降機構回原點逾時
      OUT     L4316  ; 出料托框昇降機構回原點
      OUT     T4066 K150  ; 出料托框昇降機構回原點逾時
      MPP
      LD      L4316  ; 出料托框昇降機構回原點
      AND     SM412  ; 1.0 Sec Clock
      OR      L4786  ; 出料托框昇降機構原點
      ANB
      OUT     M1066  ; 出料托框昇降機構回原點燈
      OUT     M1067  ; 出料回流機構回原點燈
4921  RET
; ----------出料開框機構-----------
      P1060
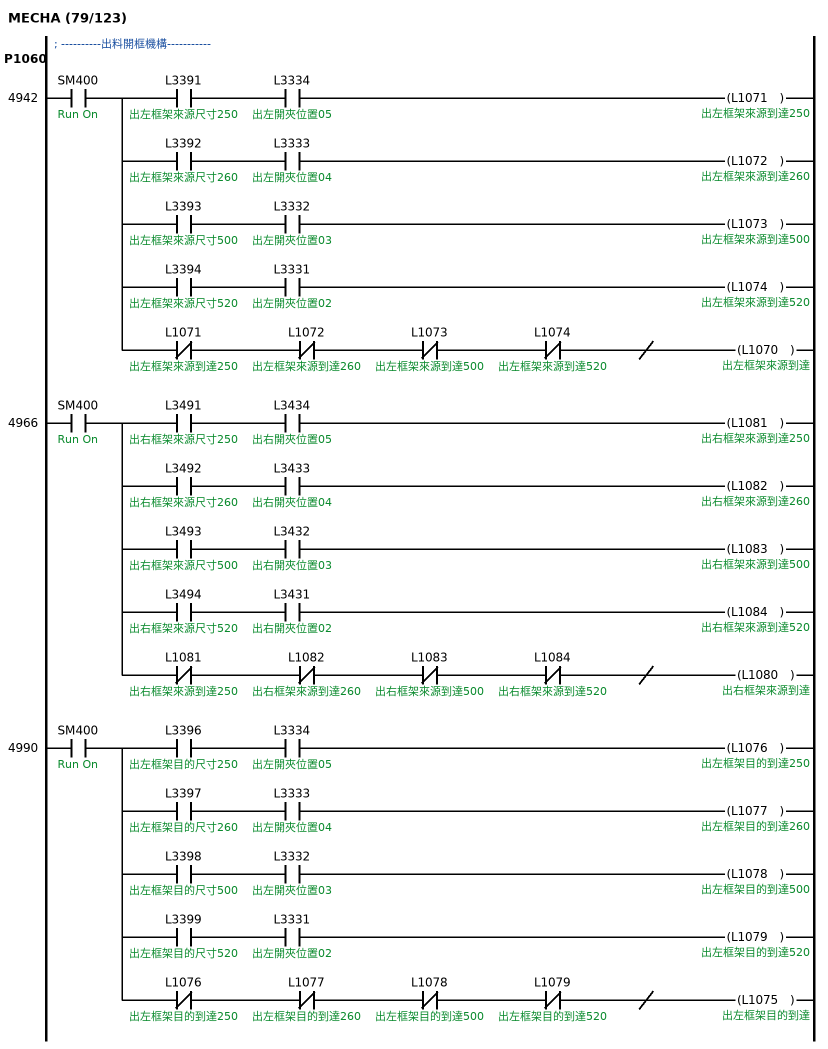
4942  LD      SM400  ; Run On
      MPS
      AND     L3391  ; 出左框架來源尺寸250
      AND     L3334  ; 出左開夾位置05
      OUT     L1071  ; 出左框架來源到達250
      MRD
      AND     L3392  ; 出左框架來源尺寸260
      AND     L3333  ; 出左開夾位置04
      OUT     L1072  ; 出左框架來源到達260
      MRD
      AND     L3393  ; 出左框架來源尺寸500
      AND     L3332  ; 出左開夾位置03
      OUT     L1073  ; 出左框架來源到達500
      MRD
      AND     L3394  ; 出左框架來源尺寸520
      AND     L3331  ; 出左開夾位置02
      OUT     L1074  ; 出左框架來源到達520
      MPP
      ANI     L1071  ; 出左框架來源到達250
      ANI     L1072  ; 出左框架來源到達260
      ANI     L1073  ; 出左框架來源到達500
      ANI     L1074  ; 出左框架來源到達520
      INV
      OUT     L1070  ; 出左框架來源到達
4966  LD      SM400  ; Run On
      MPS
      AND     L3491  ; 出右框架來源尺寸250
      AND     L3434  ; 出右開夾位置05
      OUT     L1081  ; 出右框架來源到達250
      MRD
      AND     L3492  ; 出右框架來源尺寸260
      AND     L3433  ; 出右開夾位置04
      OUT     L1082  ; 出右框架來源到達260
      MRD
      AND     L3493  ; 出右框架來源尺寸500
      AND     L3432  ; 出右開夾位置03
      OUT     L1083  ; 出右框架來源到達500
      MRD
      AND     L3494  ; 出右框架來源尺寸520
      AND     L3431  ; 出右開夾位置02
      OUT     L1084  ; 出右框架來源到達520
      MPP
      ANI     L1081  ; 出右框架來源到達250
      ANI     L1082  ; 出右框架來源到達260
      ANI     L1083  ; 出右框架來源到達500
      ANI     L1084  ; 出右框架來源到達520
      INV
      OUT     L1080  ; 出右框架來源到達
4990  LD      SM400  ; Run On
      MPS
      AND     L3396  ; 出左框架目的尺寸250
      AND     L3334  ; 出左開夾位置05
      OUT     L1076  ; 出左框架目的到達250
      MRD
      AND     L3397  ; 出左框架目的尺寸260
      AND     L3333  ; 出左開夾位置04
      OUT     L1077  ; 出左框架目的到達260
      MRD
      AND     L3398  ; 出左框架目的尺寸500
      AND     L3332  ; 出左開夾位置03
      OUT     L1078  ; 出左框架目的到達500
      MRD
      AND     L3399  ; 出左框架目的尺寸520
      AND     L3331  ; 出左開夾位置02
      OUT     L1079  ; 出左框架目的到達520
      MPP
      ANI     L1076  ; 出左框架目的到達250
      ANI     L1077  ; 出左框架目的到達260
      ANI     L1078  ; 出左框架目的到達500
      ANI     L1079  ; 出左框架目的到達520
      INV
      OUT     L1075  ; 出左框架目的到達
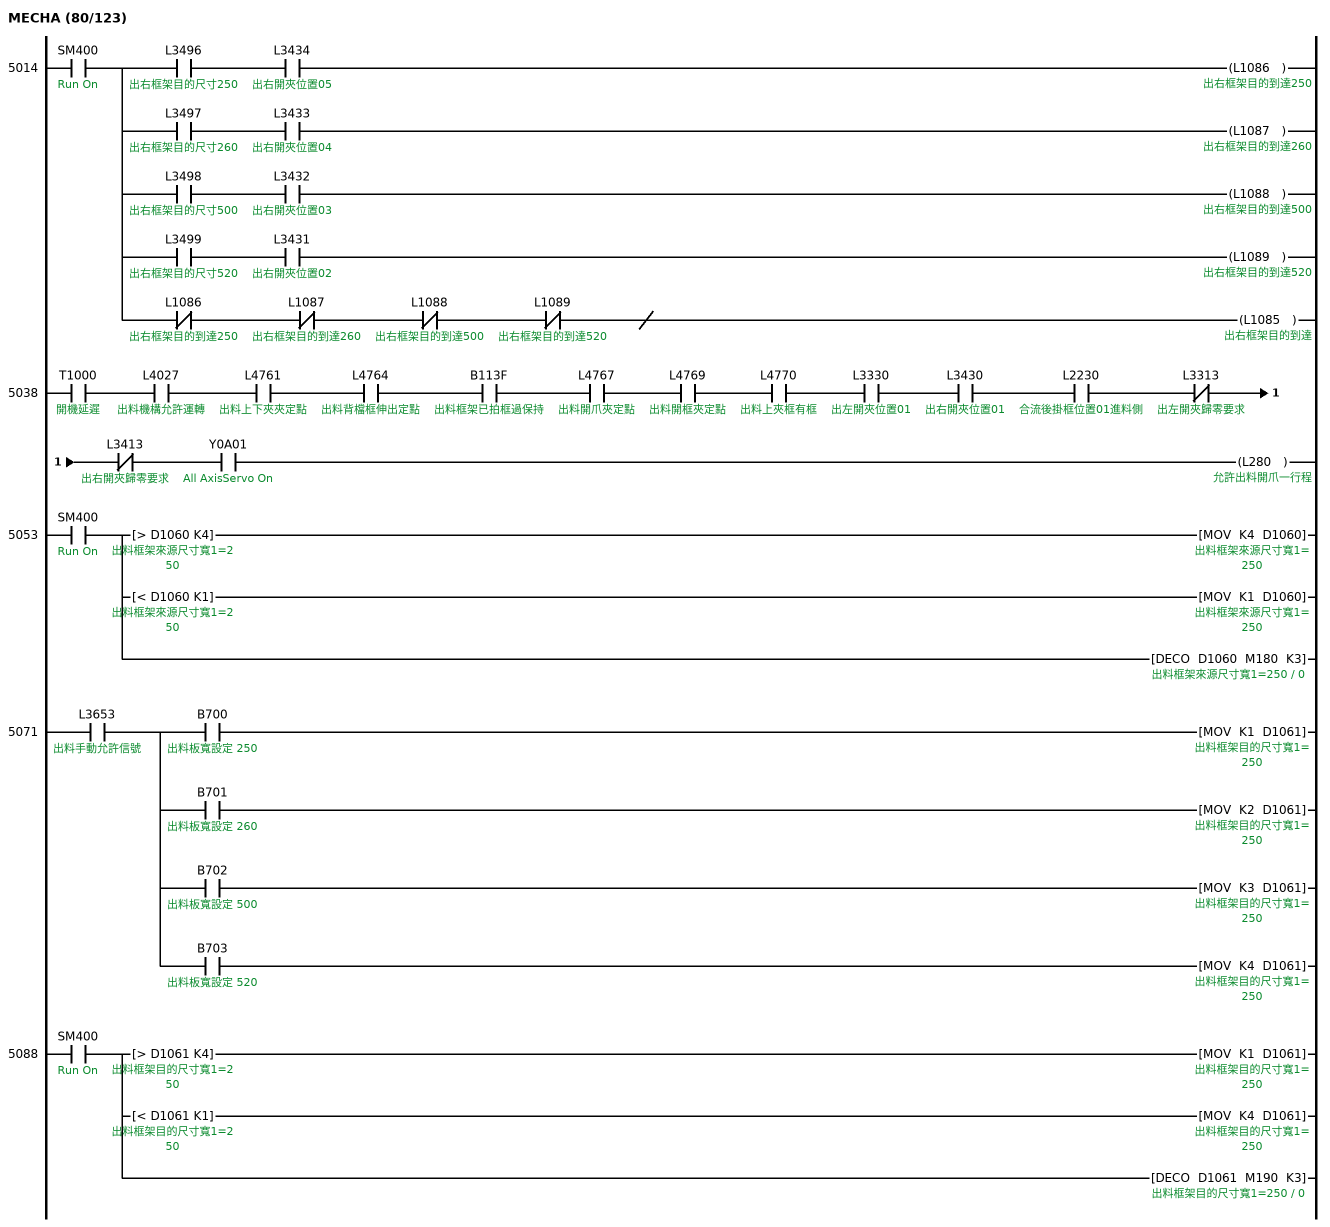
5014  LD      SM400  ; Run On
      MPS
      AND     L3496  ; 出右框架目的尺寸250
      AND     L3434  ; 出右開夾位置05
      OUT     L1086  ; 出右框架目的到達250
      MRD
      AND     L3497  ; 出右框架目的尺寸260
      AND     L3433  ; 出右開夾位置04
      OUT     L1087  ; 出右框架目的到達260
      MRD
      AND     L3498  ; 出右框架目的尺寸500
      AND     L3432  ; 出右開夾位置03
      OUT     L1088  ; 出右框架目的到達500
      MRD
      AND     L3499  ; 出右框架目的尺寸520
      AND     L3431  ; 出右開夾位置02
      OUT     L1089  ; 出右框架目的到達520
      MPP
      ANI     L1086  ; 出右框架目的到達250
      ANI     L1087  ; 出右框架目的到達260
      ANI     L1088  ; 出右框架目的到達500
      ANI     L1089  ; 出右框架目的到達520
      INV
      OUT     L1085  ; 出右框架目的到達
5038  LD      T1000  ; 開機延遲
      AND     L4027  ; 出料機構允許運轉
      AND     L4761  ; 出料上下夾夾定點
      AND     L4764  ; 出料背檔框伸出定點
      AND     B113F  ; 出料框架已拍框過保持
      AND     L4767  ; 出料開爪夾定點
      AND     L4769  ; 出料開框夾定點
      AND     L4770  ; 出料上夾框有框
      AND     L3330  ; 出左開夾位置01
      AND     L3430  ; 出右開夾位置01
      AND     L2230  ; 合流後掛框位置01進料側
      ANI     L3313  ; 出左開夾歸零要求
      ANI     L3413  ; 出右開夾歸零要求
      AND     Y0A01  ; All AxisServo On
      OUT     L280  ; 允許出料開爪一行程
5053  LD      SM400  ; Run On
      MPS
      AND>    D1060 K4  ; 出料框架來源尺寸寬1=250
      MOV     K4 D1060
      MRD
      AND<    D1060 K1  ; 出料框架來源尺寸寬1=250
      MOV     K1 D1060
      MPP
      DECO    D1060 M180 K3  ; 0
5071  LD      L3653  ; 出料手動允許信號
      MPS
      AND     B700  ; 出料板寬設定 250
      MOV     K1 D1061  ; 出料框架目的尺寸寬1=250
      MRD
      AND     B701  ; 出料板寬設定 260
      MOV     K2 D1061
      MRD
      AND     B702  ; 出料板寬設定 500
      MOV     K3 D1061
      MPP
      AND     B703  ; 出料板寬設定 520
      MOV     K4 D1061
5088  LD      SM400  ; Run On
      MPS
      AND>    D1061 K4  ; 出料框架目的尺寸寬1=250
      MOV     K1 D1061
      MRD
      AND<    D1061 K1  ; 出料框架目的尺寸寬1=250
      MOV     K4 D1061
      MPP
      DECO    D1061 M190 K3  ; 0
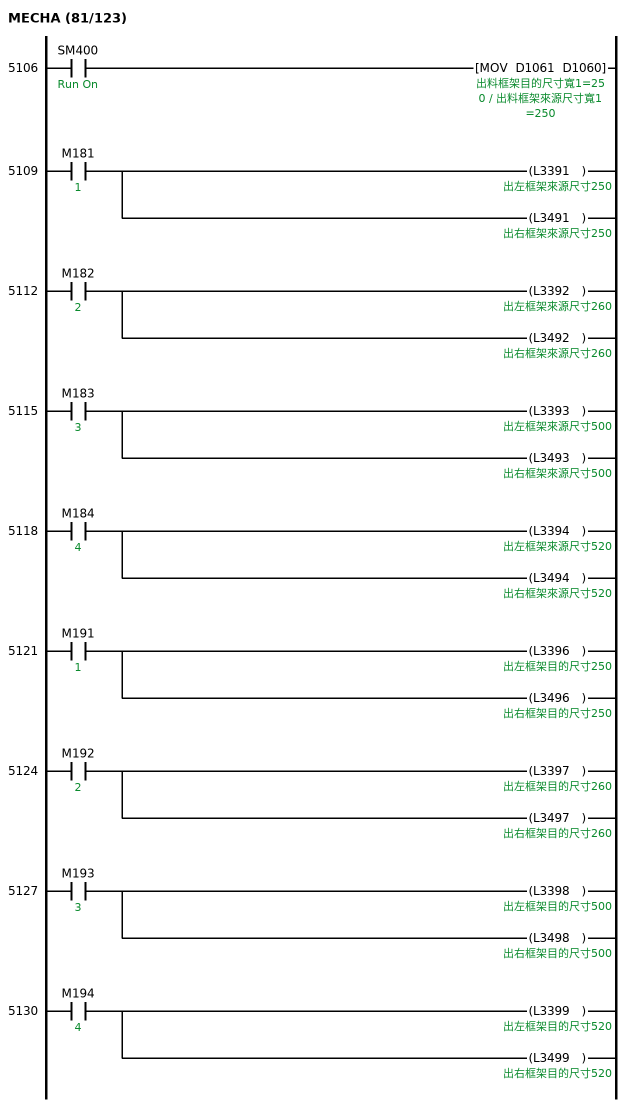
5106  LD      SM400  ; Run On
      MOV     D1061 D1060
5109  LD      M181  ; 1
      OUT     L3391  ; 出左框架來源尺寸250
      OUT     L3491  ; 出右框架來源尺寸250
5112  LD      M182  ; 2
      OUT     L3392  ; 出左框架來源尺寸260
      OUT     L3492  ; 出右框架來源尺寸260
5115  LD      M183  ; 3
      OUT     L3393  ; 出左框架來源尺寸500
      OUT     L3493  ; 出右框架來源尺寸500
5118  LD      M184  ; 4
      OUT     L3394  ; 出左框架來源尺寸520
      OUT     L3494  ; 出右框架來源尺寸520
5121  LD      M191  ; 1
      OUT     L3396  ; 出左框架目的尺寸250
      OUT     L3496  ; 出右框架目的尺寸250
5124  LD      M192  ; 2
      OUT     L3397  ; 出左框架目的尺寸260
      OUT     L3497  ; 出右框架目的尺寸260
5127  LD      M193  ; 3
      OUT     L3398  ; 出左框架目的尺寸500
      OUT     L3498  ; 出右框架目的尺寸500
5130  LD      M194  ; 4
      OUT     L3399  ; 出左框架目的尺寸520
      OUT     L3499  ; 出右框架目的尺寸520
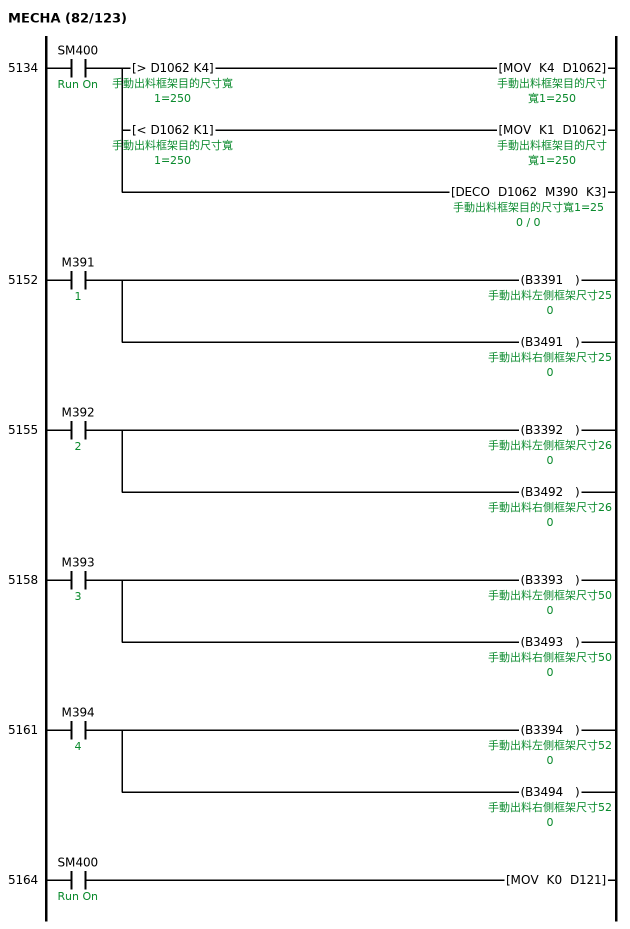
5134  LD      SM400  ; Run On
      MPS
      AND>    D1062 K4  ; 手動出料框架目的尺寸寬1=250
      MOV     K4 D1062
      MRD
      AND<    D1062 K1  ; 手動出料框架目的尺寸寬1=250
      MOV     K1 D1062
      MPP
      DECO    D1062 M390 K3  ; 0
5152  LD      M391  ; 1
      OUT     B3391  ; 手動出料左側框架尺寸250
      OUT     B3491  ; 手動出料右側框架尺寸250
5155  LD      M392  ; 2
      OUT     B3392  ; 手動出料左側框架尺寸260
      OUT     B3492  ; 手動出料右側框架尺寸260
5158  LD      M393  ; 3
      OUT     B3393  ; 手動出料左側框架尺寸500
      OUT     B3493  ; 手動出料右側框架尺寸500
5161  LD      M394  ; 4
      OUT     B3394  ; 手動出料左側框架尺寸520
      OUT     B3494  ; 手動出料右側框架尺寸520
5164  LD      SM400  ; Run On
      MOV     K0 D121
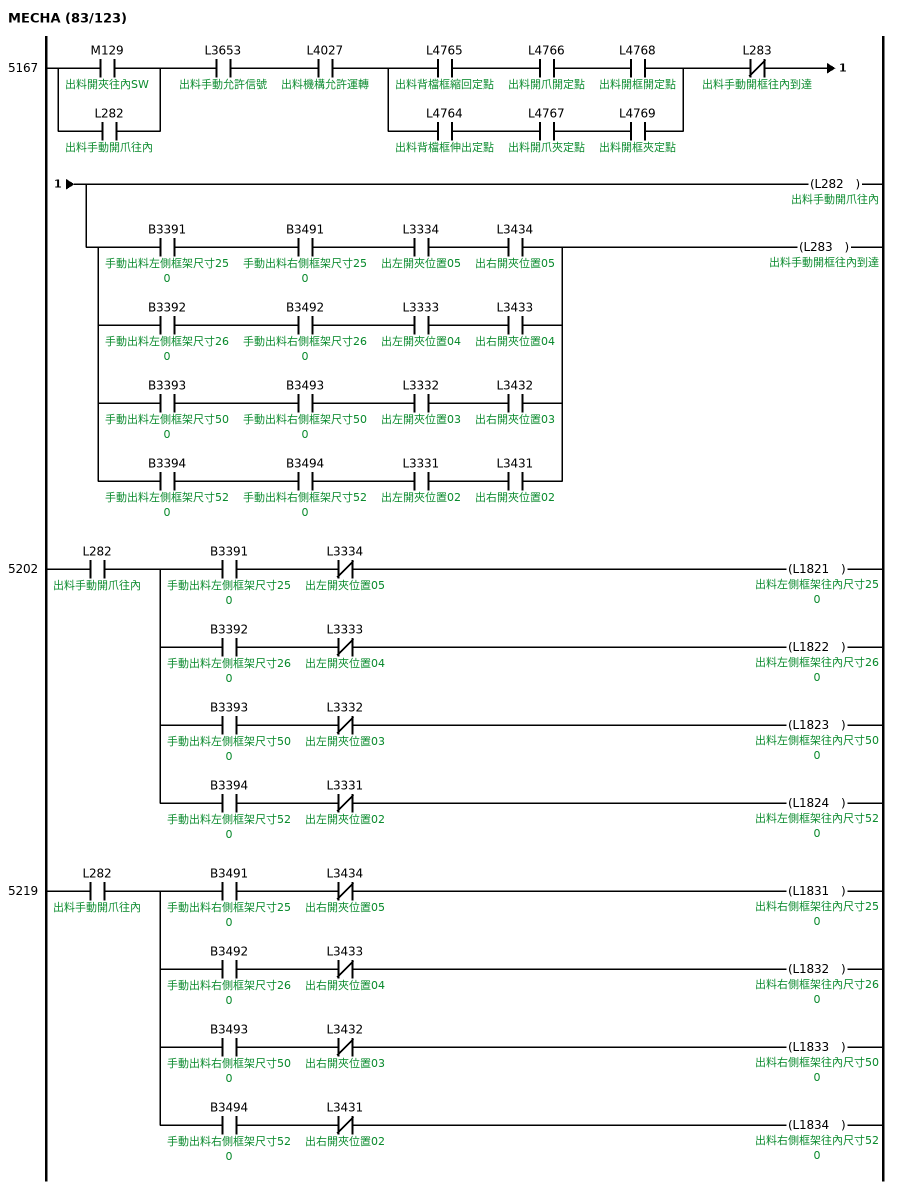
5167  LD      M129  ; 出料開夾往內SW
      OR      L282  ; 出料手動開爪往內
      AND     L3653  ; 出料手動允許信號
      AND     L4027  ; 出料機構允許運轉
      LD      L4765  ; 出料背檔框縮回定點
      AND     L4766  ; 出料開爪開定點
      AND     L4768  ; 出料開框開定點
      LD      L4764  ; 出料背檔框伸出定點
      AND     L4767  ; 出料開爪夾定點
      AND     L4769  ; 出料開框夾定點
      ORB
      ANB
      ANI     L283  ; 出料手動開框往內到達
      OUT     L282  ; 出料手動開爪往內
      LD      B3391  ; 手動出料左側框架尺寸250
      AND     B3491  ; 手動出料右側框架尺寸250
      AND     L3334  ; 出左開夾位置05
      AND     L3434  ; 出右開夾位置05
      LD      B3392  ; 手動出料左側框架尺寸260
      AND     B3492  ; 手動出料右側框架尺寸260
      AND     L3333  ; 出左開夾位置04
      AND     L3433  ; 出右開夾位置04
      ORB
      LD      B3393  ; 手動出料左側框架尺寸500
      AND     B3493  ; 手動出料右側框架尺寸500
      AND     L3332  ; 出左開夾位置03
      AND     L3432  ; 出右開夾位置03
      ORB
      LD      B3394  ; 手動出料左側框架尺寸520
      AND     B3494  ; 手動出料右側框架尺寸520
      AND     L3331  ; 出左開夾位置02
      AND     L3431  ; 出右開夾位置02
      ORB
      ANB
      OUT     L283  ; 出料手動開框往內到達
5202  LD      L282  ; 出料手動開爪往內
      MPS
      AND     B3391  ; 手動出料左側框架尺寸250
      ANI     L3334  ; 出左開夾位置05
      OUT     L1821  ; 出料左側框架往內尺寸250
      MRD
      AND     B3392  ; 手動出料左側框架尺寸260
      ANI     L3333  ; 出左開夾位置04
      OUT     L1822  ; 出料左側框架往內尺寸260
      MRD
      AND     B3393  ; 手動出料左側框架尺寸500
      ANI     L3332  ; 出左開夾位置03
      OUT     L1823  ; 出料左側框架往內尺寸500
      MPP
      AND     B3394  ; 手動出料左側框架尺寸520
      ANI     L3331  ; 出左開夾位置02
      OUT     L1824  ; 出料左側框架往內尺寸520
5219  LD      L282  ; 出料手動開爪往內
      MPS
      AND     B3491  ; 手動出料右側框架尺寸250
      ANI     L3434  ; 出右開夾位置05
      OUT     L1831  ; 出料右側框架往內尺寸250
      MRD
      AND     B3492  ; 手動出料右側框架尺寸260
      ANI     L3433  ; 出右開夾位置04
      OUT     L1832  ; 出料右側框架往內尺寸260
      MRD
      AND     B3493  ; 手動出料右側框架尺寸500
      ANI     L3432  ; 出右開夾位置03
      OUT     L1833  ; 出料右側框架往內尺寸500
      MPP
      AND     B3494  ; 手動出料右側框架尺寸520
      ANI     L3431  ; 出右開夾位置02
      OUT     L1834  ; 出料右側框架往內尺寸520
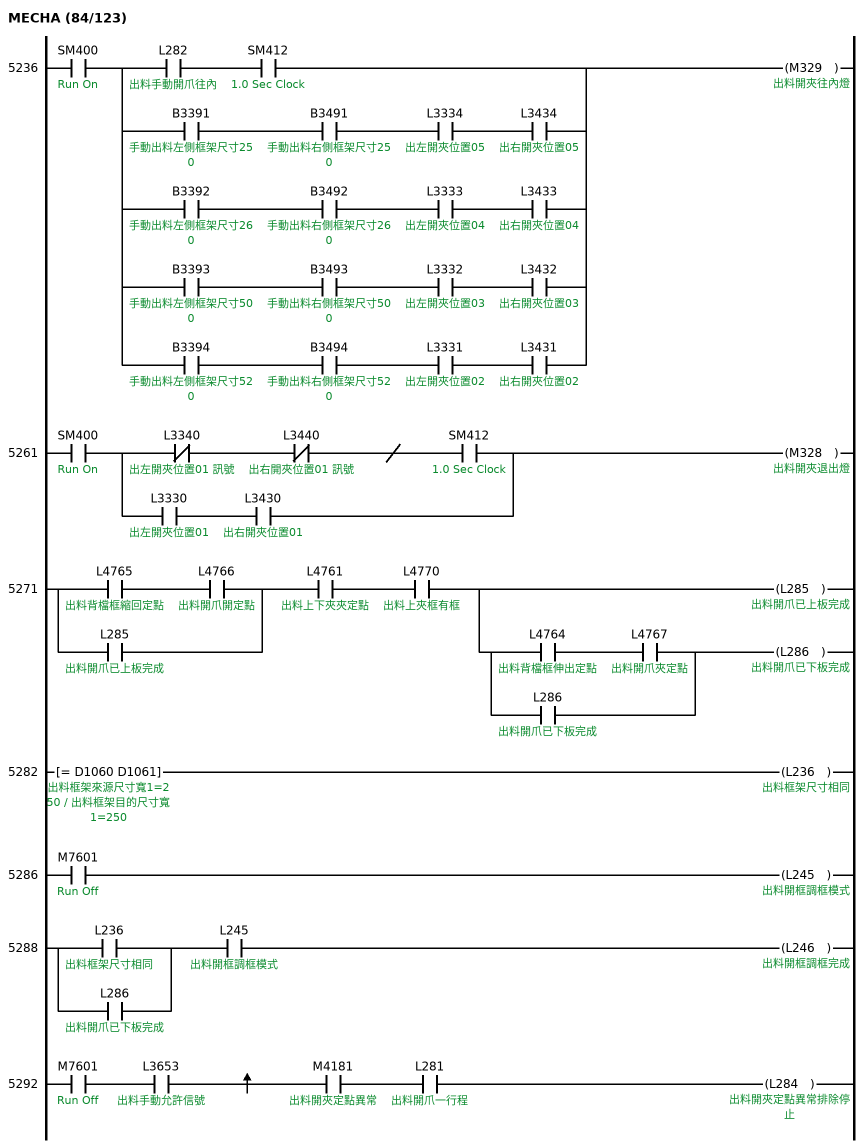
5236  LD      SM400  ; Run On
      LD      L282  ; 出料手動開爪往內
      AND     SM412  ; 1.0 Sec Clock
      LD      B3391  ; 手動出料左側框架尺寸250
      AND     B3491  ; 手動出料右側框架尺寸250
      AND     L3334  ; 出左開夾位置05
      AND     L3434  ; 出右開夾位置05
      ORB
      LD      B3392  ; 手動出料左側框架尺寸260
      AND     B3492  ; 手動出料右側框架尺寸260
      AND     L3333  ; 出左開夾位置04
      AND     L3433  ; 出右開夾位置04
      ORB
      LD      B3393  ; 手動出料左側框架尺寸500
      AND     B3493  ; 手動出料右側框架尺寸500
      AND     L3332  ; 出左開夾位置03
      AND     L3432  ; 出右開夾位置03
      ORB
      LD      B3394  ; 手動出料左側框架尺寸520
      AND     B3494  ; 手動出料右側框架尺寸520
      AND     L3331  ; 出左開夾位置02
      AND     L3431  ; 出右開夾位置02
      ORB
      ANB
      OUT     M329  ; 出料開夾往內燈
5261  LD      SM400  ; Run On
      LDI     L3340  ; 出左開夾位置01 訊號
      ANI     L3440  ; 出右開夾位置01 訊號
      INV
      AND     SM412  ; 1.0 Sec Clock
      LD      L3330  ; 出左開夾位置01
      AND     L3430  ; 出右開夾位置01
      ORB
      ANB
      OUT     M328  ; 出料開夾退出燈
5271  LD      L4765  ; 出料背檔框縮回定點
      AND     L4766  ; 出料開爪開定點
      OR      L285  ; 出料開爪已上板完成
      AND     L4761  ; 出料上下夾夾定點
      AND     L4770  ; 出料上夾框有框
      OUT     L285  ; 出料開爪已上板完成
      LD      L4764  ; 出料背檔框伸出定點
      AND     L4767  ; 出料開爪夾定點
      OR      L286  ; 出料開爪已下板完成
      ANB
      OUT     L286  ; 出料開爪已下板完成
5282  LD=     D1060 D1061  ; 出料框架來源尺寸寬1=250 / 出料框架目的尺寸寬1=250
      OUT     L236  ; 出料框架尺寸相同
5286  LD      M7601  ; Run Off
      OUT     L245  ; 出料開框調框模式
5288  LD      L236  ; 出料框架尺寸相同
      OR      L286  ; 出料開爪已下板完成
      AND     L245  ; 出料開框調框模式
      OUT     L246  ; 出料開框調框完成
5292  LD      M7601  ; Run Off
      AND     L3653  ; 出料手動允許信號
      MEP
      AND     M4181  ; 出料開夾定點異常
      AND     L281  ; 出料開爪一行程
      OUT     L284  ; 出料開夾定點異常排除停止
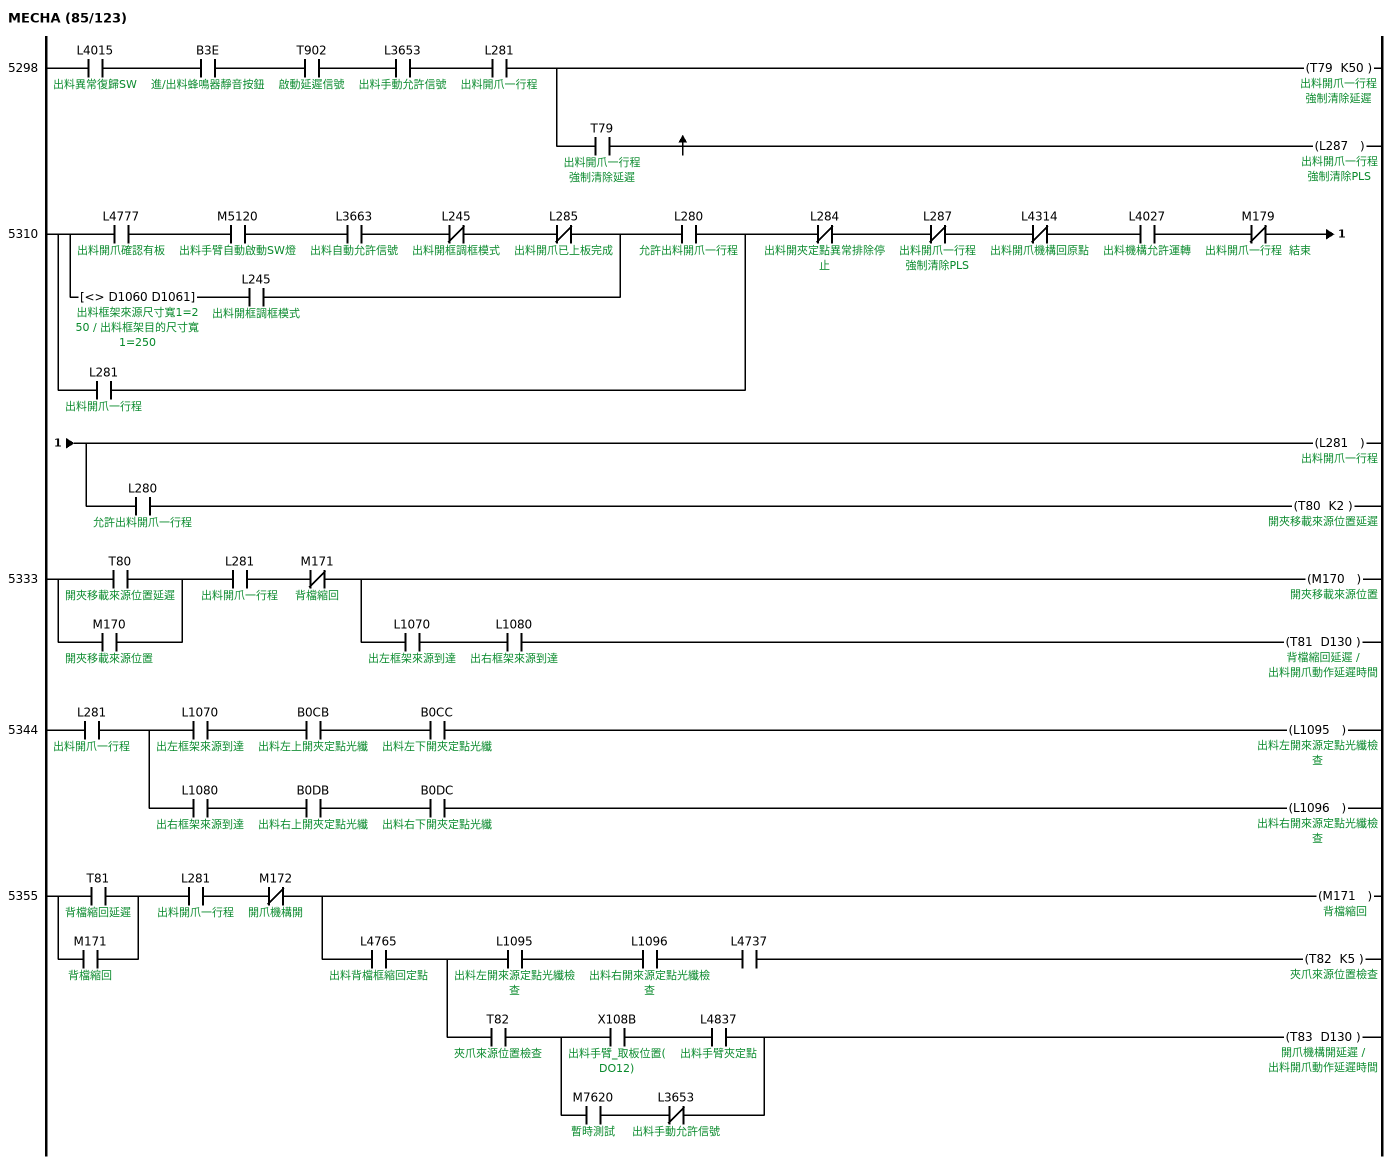
5298  LD      L4015  ; 出料異常復歸SW
      AND     B3E  ; 進/出料蜂鳴器靜音按鈕
      AND     T902  ; 啟動延遲信號
      AND     L3653  ; 出料手動允許信號
      AND     L281  ; 出料開爪一行程
      OUT     T79 K50  ; 出料開爪一行程  強制清除延遲
      AND     T79  ; 出料開爪一行程  強制清除延遲
      MEP
      OUT     L287  ; 出料開爪一行程  強制清除PLS
5310  LD      L4777  ; 出料開爪確認有板
      AND     M5120  ; 出料手臂自動啟動SW燈
      AND     L3663  ; 出料自動允許信號
      ANI     L245  ; 出料開框調框模式
      ANI     L285  ; 出料開爪已上板完成
      LD<>    D1060 D1061  ; 出料框架來源尺寸寬1=250 / 出料框架目的尺寸寬1=250
      AND     L245  ; 出料開框調框模式
      ORB
      AND     L280  ; 允許出料開爪一行程
      OR      L281  ; 出料開爪一行程
      ANI     L284  ; 出料開夾定點異常排除停止
      ANI     L287  ; 出料開爪一行程  強制清除PLS
      ANI     L4314  ; 出料開爪機構回原點
      AND     L4027  ; 出料機構允許運轉
      ANI     M179  ; 出料開爪一行程  結束
      OUT     L281  ; 出料開爪一行程
      AND     L280  ; 允許出料開爪一行程
      OUT     T80 K2  ; 開夾移載來源位置延遲
5333  LD      T80  ; 開夾移載來源位置延遲
      OR      M170  ; 開夾移載來源位置
      AND     L281  ; 出料開爪一行程
      ANI     M171  ; 背檔縮回
      OUT     M170  ; 開夾移載來源位置
      AND     L1070  ; 出左框架來源到達
      AND     L1080  ; 出右框架來源到達
      OUT     T81 D130  ; 背檔縮回延遲 / 出料開爪動作延遲時間
5344  LD      L281  ; 出料開爪一行程
      MPS
      AND     L1070  ; 出左框架來源到達
      AND     B0CB  ; 出料左上開夾定點光纖
      AND     B0CC  ; 出料左下開夾定點光纖
      OUT     L1095  ; 出料左開來源定點光纖檢查
      MPP
      AND     L1080  ; 出右框架來源到達
      AND     B0DB  ; 出料右上開夾定點光纖
      AND     B0DC  ; 出料右下開夾定點光纖
      OUT     L1096  ; 出料右開來源定點光纖檢查
5355  LD      T81  ; 背檔縮回延遲
      OR      M171  ; 背檔縮回
      AND     L281  ; 出料開爪一行程
      ANI     M172  ; 開爪機構開
      OUT     M171  ; 背檔縮回
      AND     L4765  ; 出料背檔框縮回定點
      MPS
      AND     L1095  ; 出料左開來源定點光纖檢查
      AND     L1096  ; 出料右開來源定點光纖檢查
      AND     L4737
      OUT     T82 K5  ; 夾爪來源位置檢查
      MPP
      AND     T82  ; 夾爪來源位置檢查
      LD      X108B  ; 出料手臂_取板位置(DO12)
      AND     L4837  ; 出料手臂夾定點
      LD      M7620  ; 暫時測試
      ANI     L3653  ; 出料手動允許信號
      ORB
      ANB
      OUT     T83 D130  ; 開爪機構開延遲 / 出料開爪動作延遲時間
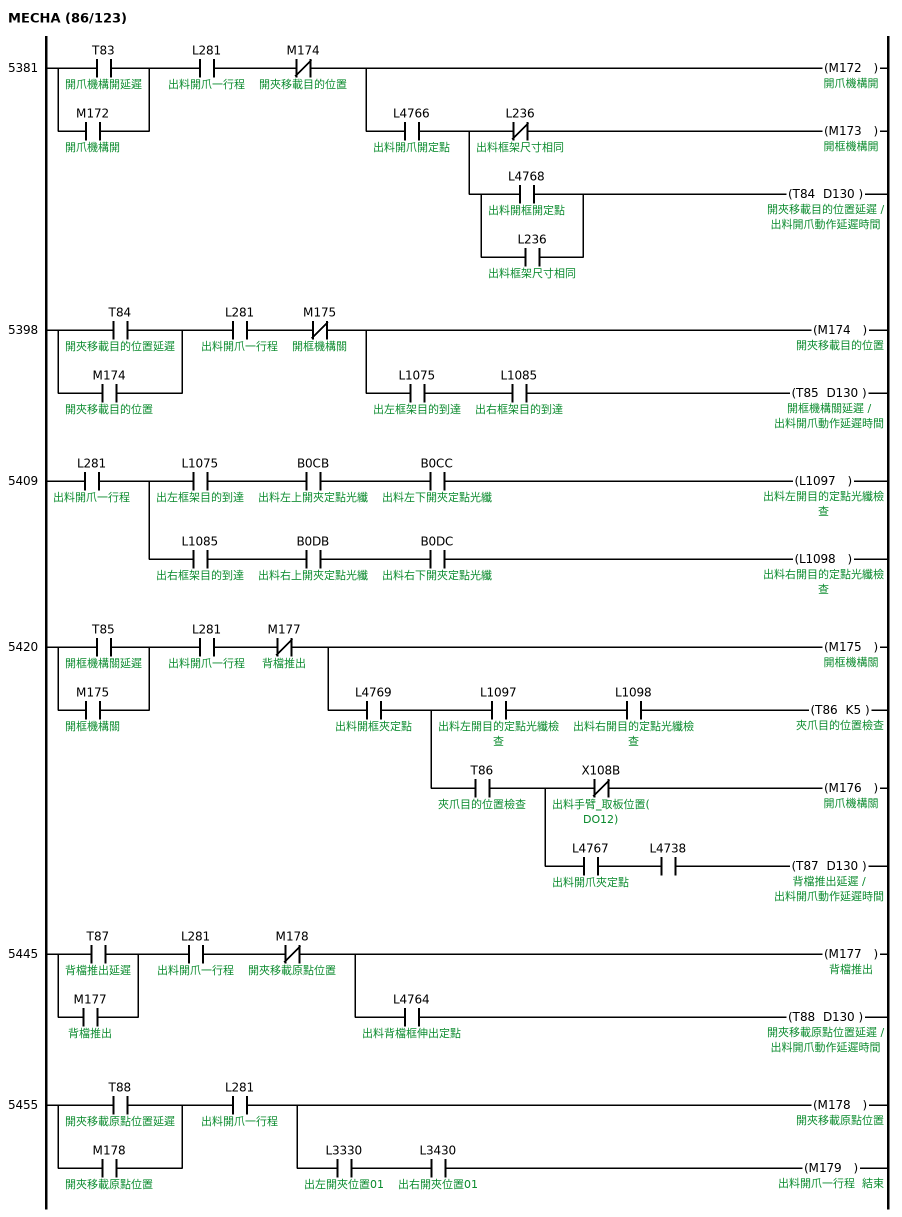
5381  LD      T83  ; 開爪機構開延遲
      OR      M172  ; 開爪機構開
      AND     L281  ; 出料開爪一行程
      ANI     M174  ; 開夾移載目的位置
      OUT     M172  ; 開爪機構開
      AND     L4766  ; 出料開爪開定點
      MPS
      ANI     L236  ; 出料框架尺寸相同
      OUT     M173  ; 開框機構開
      MPP
      LD      L4768  ; 出料開框開定點
      OR      L236  ; 出料框架尺寸相同
      ANB
      OUT     T84 D130  ; 開夾移載目的位置延遲 / 出料開爪動作延遲時間
5398  LD      T84  ; 開夾移載目的位置延遲
      OR      M174  ; 開夾移載目的位置
      AND     L281  ; 出料開爪一行程
      ANI     M175  ; 開框機構關
      OUT     M174  ; 開夾移載目的位置
      AND     L1075  ; 出左框架目的到達
      AND     L1085  ; 出右框架目的到達
      OUT     T85 D130  ; 開框機構關延遲 / 出料開爪動作延遲時間
5409  LD      L281  ; 出料開爪一行程
      MPS
      AND     L1075  ; 出左框架目的到達
      AND     B0CB  ; 出料左上開夾定點光纖
      AND     B0CC  ; 出料左下開夾定點光纖
      OUT     L1097  ; 出料左開目的定點光纖檢查
      MPP
      AND     L1085  ; 出右框架目的到達
      AND     B0DB  ; 出料右上開夾定點光纖
      AND     B0DC  ; 出料右下開夾定點光纖
      OUT     L1098  ; 出料右開目的定點光纖檢查
5420  LD      T85  ; 開框機構關延遲
      OR      M175  ; 開框機構關
      AND     L281  ; 出料開爪一行程
      ANI     M177  ; 背檔推出
      OUT     M175  ; 開框機構關
      AND     L4769  ; 出料開框夾定點
      MPS
      AND     L1097  ; 出料左開目的定點光纖檢查
      AND     L1098  ; 出料右開目的定點光纖檢查
      OUT     T86 K5  ; 夾爪目的位置檢查
      MPP
      AND     T86  ; 夾爪目的位置檢查
      MPS
      ANI     X108B  ; 出料手臂_取板位置(DO12)
      OUT     M176  ; 開爪機構關
      MPP
      AND     L4767  ; 出料開爪夾定點
      AND     L4738
      OUT     T87 D130  ; 背檔推出延遲 / 出料開爪動作延遲時間
5445  LD      T87  ; 背檔推出延遲
      OR      M177  ; 背檔推出
      AND     L281  ; 出料開爪一行程
      ANI     M178  ; 開夾移載原點位置
      OUT     M177  ; 背檔推出
      AND     L4764  ; 出料背檔框伸出定點
      OUT     T88 D130  ; 開夾移載原點位置延遲 / 出料開爪動作延遲時間
5455  LD      T88  ; 開夾移載原點位置延遲
      OR      M178  ; 開夾移載原點位置
      AND     L281  ; 出料開爪一行程
      OUT     M178  ; 開夾移載原點位置
      AND     L3330  ; 出左開夾位置01
      AND     L3430  ; 出右開夾位置01
      OUT     M179  ; 出料開爪一行程  結束
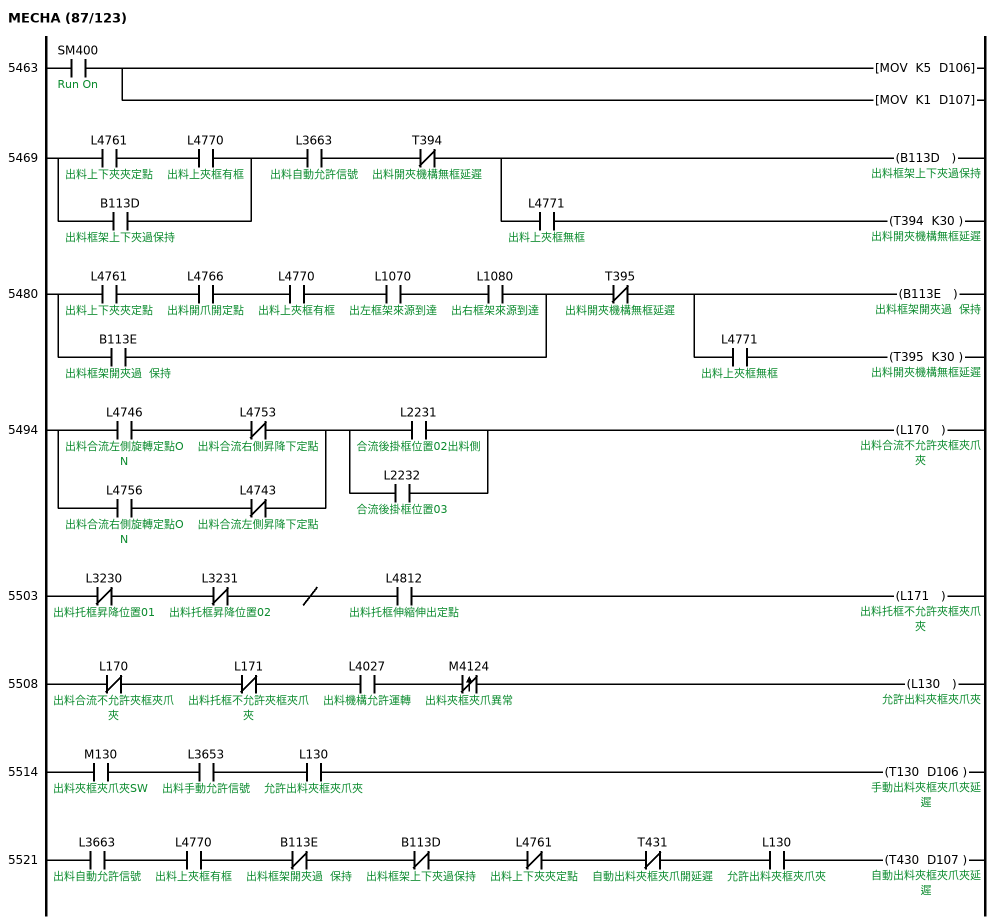
5463  LD      SM400  ; Run On
      MOV     K5 D106
      MOV     K1 D107
5469  LD      L4761  ; 出料上下夾夾定點
      AND     L4770  ; 出料上夾框有框
      OR      B113D  ; 出料框架上下夾過保持
      AND     L3663  ; 出料自動允許信號
      ANI     T394  ; 出料開夾機構無框延遲
      OUT     B113D  ; 出料框架上下夾過保持
      AND     L4771  ; 出料上夾框無框
      OUT     T394 K30  ; 出料開夾機構無框延遲
5480  LD      L4761  ; 出料上下夾夾定點
      AND     L4766  ; 出料開爪開定點
      AND     L4770  ; 出料上夾框有框
      AND     L1070  ; 出左框架來源到達
      AND     L1080  ; 出右框架來源到達
      OR      B113E  ; 出料框架開夾過  保持
      ANI     T395  ; 出料開夾機構無框延遲
      OUT     B113E  ; 出料框架開夾過  保持
      AND     L4771  ; 出料上夾框無框
      OUT     T395 K30  ; 出料開夾機構無框延遲
5494  LD      L4746  ; 出料合流左側旋轉定點ON
      ANI     L4753  ; 出料合流右側昇降下定點
      LD      L4756  ; 出料合流右側旋轉定點ON
      ANI     L4743  ; 出料合流左側昇降下定點
      ORB
      LD      L2231  ; 合流後掛框位置02出料側
      OR      L2232  ; 合流後掛框位置03
      ANB
      OUT     L170  ; 出料合流不允許夾框夾爪夾
5503  LDI     L3230  ; 出料托框昇降位置01
      ANI     L3231  ; 出料托框昇降位置02
      INV
      AND     L4812  ; 出料托框伸縮伸出定點
      OUT     L171  ; 出料托框不允許夾框夾爪夾
5508  LDI     L170  ; 出料合流不允許夾框夾爪夾
      ANI     L171  ; 出料托框不允許夾框夾爪夾
      AND     L4027  ; 出料機構允許運轉
      ANDPI   M4124  ; 出料夾框夾爪異常
      OUT     L130  ; 允許出料夾框夾爪夾
5514  LD      M130  ; 出料夾框夾爪夾SW
      AND     L3653  ; 出料手動允許信號
      AND     L130  ; 允許出料夾框夾爪夾
      OUT     T130 D106  ; 手動出料夾框夾爪夾延遲
5521  LD      L3663  ; 出料自動允許信號
      AND     L4770  ; 出料上夾框有框
      ANI     B113E  ; 出料框架開夾過  保持
      ANI     B113D  ; 出料框架上下夾過保持
      ANI     L4761  ; 出料上下夾夾定點
      ANI     T431  ; 自動出料夾框夾爪開延遲
      AND     L130  ; 允許出料夾框夾爪夾
      OUT     T430 D107  ; 自動出料夾框夾爪夾延遲
